HMI tags "2080AG504M01"
   "2080AG504M01.AI1" : Real AT %DB4149.DBD6, 500 ms
   "2080AG504M01.AI2" : Real AT %DB4149.DBD10, 500 ms
   "2080AG504M01.AI3" : Real AT %DB4149.DBD14, 500 ms
   "2080AG504M01.AO1a" : Real AT %DB4149.DBD34, 500 ms
   "2080AG504M01.AO1b" : Real AT %DB4149.DBD38, 500 ms
   "2080AG504M01.AO2a" : Real AT %DB4149.DBD42, 500 ms
   "2080AG504M01.AO2b" : Real AT %DB4149.DBD42, 500 ms
   "2080AG504M01.AO3a" : Real AT %DB4149.DBD50, 500 ms
   "2080AG504M01.AO3b" : Real AT %DB4149.DBD46, 500 ms
   "2080AG504M01.BlockInfo" : Array [0..4] of Int AT %DB4149.DBX74.0, 500 ms
   "2080AG504M01.DefaultText" : TextRef, internal   // Заголовок POPUP окна. При експорте из ECS через скрипт заполняется автоматически, если теги копируются в ручную то требуется в ручную задатать свойство Start Value
   "2080AG504M01.DI.ACK" : Bool AT %DB4149.DBX5.3, 500 ms
   "2080AG504M01.DI.ASTR" : Bool AT %DB4149.DBX2.1, 500 ms
   "2080AG504M01.DI.BUSF" : Bool AT %DB4149.DBX4.5, 500 ms
   "2080AG504M01.DI.DIR" : Bool AT %DB4149.DBX2.2, 500 ms
   "2080AG504M01.DI.DOPR" : Bool AT %DB4149.DBX4.6, 500 ms
   "2080AG504M01.DI.DRDY" : Bool AT %DB4149.DBX3.6, 500 ms
   "2080AG504M01.DI.DTEST" : Bool AT %DB4149.DBX4.7, 500 ms
   "2080AG504M01.DI.EARTH" : Bool AT %DB4149.DBX4.1, 500 ms
   "2080AG504M01.DI.ES" : Bool AT %DB4149.DBX5.2, 500 ms
   "2080AG504M01.DI.GFA" : Bool AT %DB4149.DBX4.3, 500 ms
   "2080AG504M01.DI.GWA" : Bool AT %DB4149.DBX4.4, 500 ms
   "2080AG504M01.DI.LSTP" : Bool AT %DB4149.DBX3.2, 500 ms
   "2080AG504M01.DI.LSTR1" : Bool AT %DB4149.DBX3.0, 500 ms
   "2080AG504M01.DI.LSTR2" : Bool AT %DB4149.DBX3.1, 500 ms
   "2080AG504M01.DI.MCC" : Bool AT %DB4149.DBX2.3, 500 ms
   "2080AG504M01.DI.MD" : Bool AT %DB4149.DBX3.7, 500 ms
   "2080AG504M01.DI.OVL" : Bool AT %DB4149.DBX2.5, 500 ms
   "2080AG504M01.DI.RDY" : Bool AT %DB4149.DBX2.4, 500 ms
   "2080AG504M01.DI.REM" : Bool AT %DB4149.DBX3.3, 500 ms
   "2080AG504M01.DI.RET1" : Bool AT %DB4149.DBX2.6, 500 ms
   "2080AG504M01.DI.RET2" : Bool AT %DB4149.DBX2.7, 500 ms
   "2080AG504M01.DI.SEL" : Bool AT %DB4149.DBX2.0, 500 ms
   "2080AG504M01.DI.SFS" : Bool AT %DB4149.DBX5.0, 500 ms
   "2080AG504M01.DI.SLS" : Bool AT %DB4149.DBX5.1, 500 ms
   "2080AG504M01.DI.SSW" : Bool AT %DB4149.DBX3.4, 500 ms
   "2080AG504M01.DI.STALL" : Bool AT %DB4149.DBX4.0, 500 ms
   "2080AG504M01.DI.TFA" : Bool AT %DB4149.DBX3.5, 500 ms
   "2080AG504M01.DI.UBAL" : Bool AT %DB4149.DBX4.2, 500 ms
   "2080AG504M01.DQ.ASTW" : Bool AT %DB4149.DBX32.0, 500 ms
   "2080AG504M01.DQ.AUT" : Bool AT %DB4149.DBX31.4, 500 ms
   "2080AG504M01.DQ.CON1" : Bool AT %DB4149.DBX30.0, 500 ms
   "2080AG504M01.DQ.CON2" : Bool AT %DB4149.DBX30.1, 500 ms
   "2080AG504M01.DQ.LAMP1" : Bool AT %DB4149.DBX30.2, 500 ms
   "2080AG504M01.DQ.LAMP2" : Bool AT %DB4149.DBX30.3, 500 ms
   "2080AG504M01.DQ.LOC" : Bool AT %DB4149.DBX31.2, 500 ms
   "2080AG504M01.DQ.MAN" : Bool AT %DB4149.DBX31.3, 500 ms
   "2080AG504M01.DQ.OK" : Bool AT %DB4149.DBX31.1, 500 ms
   "2080AG504M01.DQ.RD1" : Bool AT %DB4149.DBX30.5, 500 ms
   "2080AG504M01.DQ.RD2" : Bool AT %DB4149.DBX30.6, 500 ms
   "2080AG504M01.DQ.RES" : Bool AT %DB4149.DBX31.6, 500 ms
   "2080AG504M01.DQ.RUN1" : Bool AT %DB4149.DBX30.7, 500 ms
   "2080AG504M01.DQ.RUN2" : Bool AT %DB4149.DBX31.0, 500 ms
   "2080AG504M01.DQ.SACK" : Bool AT %DB4149.DBX30.4, 500 ms
   "2080AG504M01.DQ.SS" : Bool AT %DB4149.DBX31.5, 500 ms
   "2080AG504M01.DQ.TESTP" : Bool AT %DB4149.DBX31.7, 500 ms
   "2080AG504M01.FP_CMD" : Int AT %DB4149.DBW84, 500 ms
   "2080AG504M01.FP_CMD.AckAlarm" : Bool AT %DB4149.DBX84.7, 500 ms
   "2080AG504M01.FP_CMD.Auto" : Bool AT %DB4149.DBX85.0, 500 ms
   "2080AG504M01.FP_CMD.Local" : Bool AT %DB4149.DBX85.2, 500 ms
   "2080AG504M01.FP_CMD.Manual" : Bool AT %DB4149.DBX85.1, 500 ms
   "2080AG504M01.FP_CMD.QuickStop" : Bool AT %DB4149.DBX84.0, 500 ms
   "2080AG504M01.FP_CMD.Reset" : Bool AT %DB4149.DBX85.6, 500 ms
   "2080AG504M01.FP_CMD.Start1" : Bool AT %DB4149.DBX85.3, 500 ms
   "2080AG504M01.FP_CMD.Start2" : Bool AT %DB4149.DBX85.4, 500 ms
   "2080AG504M01.FP_CMD.Stop" : Bool AT %DB4149.DBX85.5, 500 ms
   "2080AG504M01.FP_CMD.Test" : Bool AT %DB4149.DBX85.7, 500 ms
   "2080AG504M01.FP_DIM.Auto" : Bool AT %DB4149.DBX92.0, 500 ms
   "2080AG504M01.FP_DIM.FP_DIM" : Bool AT %DB4149.DBX92.0, 500 ms
   "2080AG504M01.FP_DIM.Local" : Bool AT %DB4149.DBX92.1, 500 ms
   "2080AG504M01.FP_DIM.Manual" : Bool AT %DB4149.DBX92.2, 500 ms
   "2080AG504M01.FP_DIM.QStop" : Bool AT %DB4149.DBX92.7, 500 ms
   "2080AG504M01.FP_DIM.Reset" : Bool AT %DB4149.DBX93.0, 500 ms
   "2080AG504M01.FP_DIM.Start1" : Bool AT %DB4149.DBX92.3, 500 ms
   "2080AG504M01.FP_DIM.Start2" : Bool AT %DB4149.DBX92.4, 500 ms
   "2080AG504M01.FP_DIM.Stop" : Bool AT %DB4149.DBX92.5, 500 ms
   "2080AG504M01.FP_DIM.TEst" : Bool AT %DB4149.DBX92.6, 500 ms
   "2080AG504M01.FP_DIM1" : Array [0..15] of Bool AT %DB4149.DBX92.0, 500 ms
   "2080AG504M01.FP_EN.Mode_Auto" : Bool AT %DB4149.DBX90.0, 500 ms
   "2080AG504M01.FP_EN.Mode_Loc" : Bool AT %DB4149.DBX90.2, 500 ms
   "2080AG504M01.FP_EN.Mode_Loc_1" : Bool AT %DB4149.DBX90.3, 500 ms
   "2080AG504M01.FP_EN.Mode_Man" : Bool AT %DB4149.DBX90.1, 500 ms
   "2080AG504M01.FP_EN.Mode_SS_Field" : Bool AT %DB4149.DBX90.4, 500 ms
   "2080AG504M01.FP_EN.Mode_SS_FP" : Bool AT %DB4149.DBX90.5, 500 ms
   "2080AG504M01.FP_EN.Mode_Test" : Bool AT %DB4149.DBX90.3, 500 ms
   "2080AG504M01.FP_EN.PB_QStop" : Bool AT %DB4149.DBX90.6, 500 ms
   "2080AG504M01.FP_PARM.AI1_Max" : Real AT %DB4149.DBD158, 500 ms
   "2080AG504M01.FP_PARM.AI1_Min" : Real AT %DB4149.DBD162, 500 ms
   "2080AG504M01.FP_PARM.AI2_Max" : Real AT %DB4149.DBD166, 500 ms
   "2080AG504M01.FP_PARM.AI2_Min" : Real AT %DB4149.DBD170, 500 ms
   "2080AG504M01.FP_PARM.AI3_Max" : Real AT %DB4149.DBD174, 500 ms
   "2080AG504M01.FP_PARM.AI3_Min" : Real AT %DB4149.DBD178, 500 ms
   "2080AG504M01.FP_PARM.AO1a_Max" : Real AT %DB4149.DBD182, 500 ms
   "2080AG504M01.FP_PARM.AO1a_Min" : Real AT %DB4149.DBD186, 500 ms
   "2080AG504M01.FP_PARM.AO1b_Max" : Real AT %DB4149.DBD206, 500 ms
   "2080AG504M01.FP_PARM.AO1b_Min" : Real AT %DB4149.DBD210, 500 ms
   "2080AG504M01.FP_PARM.AO2a_Max" : Real AT %DB4149.DBD190, 500 ms
   "2080AG504M01.FP_PARM.AO2a_Min" : Real AT %DB4149.DBD194, 500 ms
   "2080AG504M01.FP_PARM.AO2b_Max" : Real AT %DB4149.DBD214, 500 ms
   "2080AG504M01.FP_PARM.AO2b_Min" : Real AT %DB4149.DBD218, 500 ms
   "2080AG504M01.FP_PARM.AO3a_Max" : Real AT %DB4149.DBD198, 500 ms
   "2080AG504M01.FP_PARM.AO3a_Min" : Real AT %DB4149.DBD202, 500 ms
   "2080AG504M01.FP_PARM.AO3b_Max" : Real AT %DB4149.DBD222, 500 ms
   "2080AG504M01.FP_PARM.AO3b_Min" : Real AT %DB4149.DBD226, 500 ms
   "2080AG504M01.FP_PARM.ChangeDir_Acc" : Int AT %DB4149.DBW138, 500 ms
   "2080AG504M01.FP_PARM.ChangeDir_Pre" : Int AT %DB4149.DBW136, 500 ms
   "2080AG504M01.FP_PARM.DelayStart_Acc" : Int AT %DB4149.DBW114, 500 ms
   "2080AG504M01.FP_PARM.DelayStart_Pre" : Int AT %DB4149.DBW112, 500 ms
   "2080AG504M01.FP_PARM.DelayStop_Acc" : Int AT %DB4149.DBW118, 500 ms
   "2080AG504M01.FP_PARM.DelayStop_Pre" : Int AT %DB4149.DBW116, 500 ms
   "2080AG504M01.FP_PARM.INTL" : Bool AT %DB4149.DBX230.0, 500 ms
   "2080AG504M01.FP_PARM.INTL_SEQ_STP" : Bool AT %DB4149.DBX230.3, 500 ms
   "2080AG504M01.FP_PARM.INTL_SEQ_STR1" : Bool AT %DB4149.DBX230.1, 500 ms
   "2080AG504M01.FP_PARM.INTL_SEQ_STR2" : Bool AT %DB4149.DBX230.2, 500 ms
   "2080AG504M01.FP_PARM.LeaveFS_Acc" : Int AT %DB4149.DBW142, 500 ms
   "2080AG504M01.FP_PARM.LeaveFS_Pre" : Int AT %DB4149.DBW140, 500 ms
   "2080AG504M01.FP_PARM.MD_Freq_PV" : Int AT %DB4149.DBW154, 500 ms
   "2080AG504M01.FP_PARM.MD_Freq_SP" : Int AT %DB4149.DBW152, 500 ms
   "2080AG504M01.FP_PARM.ReachFS_Acc" : Int AT %DB4149.DBW150, 500 ms
   "2080AG504M01.FP_PARM.ReachFS_Pre" : Int AT %DB4149.DBW148, 500 ms
   "2080AG504M01.FP_PARM.ReachLS_Acc" : Int AT %DB4149.DBW146, 500 ms
   "2080AG504M01.FP_PARM.ReachLS_Pre" : Int AT %DB4149.DBW144, 500 ms
   "2080AG504M01.FP_PARM.ReturnMon_Acc" : Int AT %DB4149.DBW122, 500 ms
   "2080AG504M01.FP_PARM.ReturnMon_Pre" : Int AT %DB4149.DBW120, 500 ms
   "2080AG504M01.FP_PARM.RunDelay1_Acc" : Int AT %DB4149.DBW106, 500 ms
   "2080AG504M01.FP_PARM.RunDelay1_Pre" : Int AT %DB4149.DBW104, 500 ms
   "2080AG504M01.FP_PARM.RunDelay2_Acc" : Int AT %DB4149.DBW110, 500 ms
   "2080AG504M01.FP_PARM.RunDelay2_Pre" : Int AT %DB4149.DBW108, 500 ms
   "2080AG504M01.FP_PARM.SpeedMonOffDelay_Acc" : Int AT %DB4149.DBW130, 500 ms
   "2080AG504M01.FP_PARM.SpeedMonOffDelay_Pre" : Int AT %DB4149.DBW128, 500 ms
   "2080AG504M01.FP_PARM.SpeedMonOnDelay_Acc" : Int AT %DB4149.DBW126, 500 ms
   "2080AG504M01.FP_PARM.SpeedMonOnDelay_Pre" : Int AT %DB4149.DBW124, 500 ms
   "2080AG504M01.FP_PARM.SpeedMonTrigDelay_Acc" : Int AT %DB4149.DBW134, 500 ms
   "2080AG504M01.FP_PARM.SpeedMonTrigDelay_Pre" : Int AT %DB4149.DBW132, 500 ms
   "2080AG504M01.FP_PARM.StartWarn_Acc" : Int AT %DB4149.DBW102, 500 ms
   "2080AG504M01.FP_PARM.StartWarn_Pre" : Int AT %DB4149.DBW100, 500 ms
   "2080AG504M01.FP_PARM.StopReason" : Int AT %DB4149.DBW156, 500 ms
   "2080AG504M01.FP_SEL.INCH_Loc" : Bool AT %DB4149.DBX87.7, 500 ms
   "2080AG504M01.FP_SEL.INCH_Man" : Bool AT %DB4149.DBX87.6, 500 ms
   "2080AG504M01.FP_SEL.MD" : Bool AT %DB4149.DBX86.0, 500 ms
   "2080AG504M01.FP_SEL.MD_Maintain" : Bool AT %DB4149.DBX86.3, 500 ms
   "2080AG504M01.FP_SEL.MD_OnOff" : Bool AT %DB4149.DBX86.2, 500 ms
   "2080AG504M01.FP_SEL.MD_Puls" : Bool AT %DB4149.DBX86.1, 500 ms
   "2080AG504M01.FP_SEL.MotorStarter" : Bool AT %DB4149.DBX87.3, 500 ms
   "2080AG504M01.FP_SEL.OutOfSevice" : Bool AT %DB4149.DBX88.0, 500 ms
   "2080AG504M01.FP_SEL.ParentCollection" : Bool AT %DB4149.DBX87.5, 500 ms
   "2080AG504M01.FP_SEL.ParentSupress" : Bool AT %DB4149.DBX87.4, 500 ms
   "2080AG504M01.FP_SEL.STW_AutoStart" : Bool AT %DB4149.DBX86.4, 500 ms
   "2080AG504M01.FP_SEL.STW_Local" : Bool AT %DB4149.DBX86.5, 500 ms
   "2080AG504M01.FP_SEL.STW_Manual" : Bool AT %DB4149.DBX86.6, 500 ms
   "2080AG504M01.FP_SEL.STW_Single" : Bool AT %DB4149.DBX86.7, 500 ms
   "2080AG504M01.FP_SEL.Type_Bimotor" : Bool AT %DB4149.DBX87.1, 500 ms
   "2080AG504M01.FP_SEL.Type_Indication" : Bool AT %DB4149.DBX87.2, 500 ms
   "2080AG504M01.FP_SEL.Type_Unimotor" : Bool AT %DB4149.DBX87.0, 500 ms
   "2080AG504M01.FP_SEL.WarningDrive" : Bool AT %DB4149.DBX88.1, 500 ms
   "2080AG504M01.FP_SHOW.ACK" : Bool AT %DB4149.DBX97.5, 500 ms
   "2080AG504M01.FP_SHOW.AI1" : Bool AT %DB4149.DBX95.0, 500 ms
   "2080AG504M01.FP_SHOW.AI2" : Bool AT %DB4149.DBX95.1, 500 ms
   "2080AG504M01.FP_SHOW.AI3" : Bool AT %DB4149.DBX95.2, 500 ms
   "2080AG504M01.FP_SHOW.ASTR" : Bool AT %DB4149.DBX99.2, 500 ms
   "2080AG504M01.FP_SHOW.B1" : Byte AT %DB4149.DBB95, 500 ms
   "2080AG504M01.FP_SHOW.B2" : Byte AT %DB4149.DBB96, 500 ms
   "2080AG504M01.FP_SHOW.B3" : Byte AT %DB4149.DBB97, 500 ms
   "2080AG504M01.FP_SHOW.B4" : Byte AT %DB4149.DBB98, 500 ms
   "2080AG504M01.FP_SHOW.BUSF" : Bool AT %DB4149.DBX97.2, 500 ms
   "2080AG504M01.FP_SHOW.ChangeDir" : Bool AT %DB4149.DBX99.0, 500 ms
   "2080AG504M01.FP_SHOW.CON2" : Bool AT %DB4149.DBX98.2, 500 ms
   "2080AG504M01.FP_SHOW.DelayRun2" : Bool AT %DB4149.DBX98.7, 500 ms
   "2080AG504M01.FP_SHOW.DOPR" : Bool AT %DB4149.DBX97.3, 500 ms
   "2080AG504M01.FP_SHOW.DRDY" : Bool AT %DB4149.DBX96.4, 500 ms
   "2080AG504M01.FP_SHOW.DTEST" : Bool AT %DB4149.DBX97.4, 500 ms
   "2080AG504M01.FP_SHOW.EARTH" : Bool AT %DB4149.DBX96.6, 500 ms
   "2080AG504M01.FP_SHOW.ES" : Bool AT %DB4149.DBX96.2, 500 ms
   "2080AG504M01.FP_SHOW.GFA" : Bool AT %DB4149.DBX97.0, 500 ms
   "2080AG504M01.FP_SHOW.GWA" : Bool AT %DB4149.DBX97.1, 500 ms
   "2080AG504M01.FP_SHOW.LSTP" : Bool AT %DB4149.DBX95.7, 500 ms
   "2080AG504M01.FP_SHOW.LSTR1" : Bool AT %DB4149.DBX97.6, 500 ms
   "2080AG504M01.FP_SHOW.LSTR2" : Bool AT %DB4149.DBX97.7, 500 ms
   "2080AG504M01.FP_SHOW.MCC" : Bool AT %DB4149.DBX95.4, 500 ms
   "2080AG504M01.FP_SHOW.MD" : Bool AT %DB4149.DBX98.6, 500 ms
   "2080AG504M01.FP_SHOW.OVL" : Bool AT %DB4149.DBX95.6, 500 ms
   "2080AG504M01.FP_SHOW.PB_Auto" : Bool AT %DB4149.DBX94.0, 500 ms
   "2080AG504M01.FP_SHOW.PB_Local" : Bool AT %DB4149.DBX94.1, 500 ms
   "2080AG504M01.FP_SHOW.PB_Manual" : Bool AT %DB4149.DBX94.2, 500 ms
   "2080AG504M01.FP_SHOW.PB_QStop" : Bool AT %DB4149.DBX94.7, 500 ms
   "2080AG504M01.FP_SHOW.PB_Reset" : Bool AT %DB4149.DBX99.1, 500 ms
   "2080AG504M01.FP_SHOW.PB_Start1" : Bool AT %DB4149.DBX94.3, 500 ms
   "2080AG504M01.FP_SHOW.PB_Start2" : Bool AT %DB4149.DBX94.4, 500 ms
   "2080AG504M01.FP_SHOW.PB_Stop" : Bool AT %DB4149.DBX94.5, 500 ms
   "2080AG504M01.FP_SHOW.PB_Test" : Bool AT %DB4149.DBX94.6, 500 ms
   "2080AG504M01.FP_SHOW.RD2" : Bool AT %DB4149.DBX98.3, 500 ms
   "2080AG504M01.FP_SHOW.RDY" : Bool AT %DB4149.DBX95.5, 500 ms
   "2080AG504M01.FP_SHOW.REM" : Bool AT %DB4149.DBX96.0, 500 ms
   "2080AG504M01.FP_SHOW.RET2" : Bool AT %DB4149.DBX98.0, 500 ms
   "2080AG504M01.FP_SHOW.RUN2" : Bool AT %DB4149.DBX98.1, 500 ms
   "2080AG504M01.FP_SHOW.SFS" : Bool AT %DB4149.DBX98.4, 500 ms
   "2080AG504M01.FP_SHOW.SLS" : Bool AT %DB4149.DBX98.5, 500 ms
   "2080AG504M01.FP_SHOW.SP" : Bool AT %DB4149.DBX95.3, 500 ms
   "2080AG504M01.FP_SHOW.SSW" : Bool AT %DB4149.DBX96.1, 500 ms
   "2080AG504M01.FP_SHOW.STALL" : Bool AT %DB4149.DBX96.5, 500 ms
   "2080AG504M01.FP_SHOW.TFA" : Bool AT %DB4149.DBX96.3, 500 ms
   "2080AG504M01.FP_SHOW.UBAL" : Bool AT %DB4149.DBX96.7, 500 ms
   "2080AG504M01.ModePointer" : Int AT %DB4149.DBW496, 500 ms
   "2080AG504M01.MSW" : DWord AT %DB4149.DBD62, 500 ms
   "2080AG504M01.ParentInfo" : TextRef, internal   // Имя родителя для попап окна, вкладка инфо. При експорте из ECS через скрипт заполняется автоматически, если теги копируются в ручную то требуется в ручную задатать свойство Start Value
   "2080AG504M01.SPSET" : Real AT %DB4149.DBD18, 500 ms
   "2080AG504M01.StatusWork" : Int AT %DB4149.DBW494, 500 ms
   "2080AG504M01.STR01" : Byte AT %DB10.DBB103, 500 ms   // Interlock
   "2080AG504M01.STR01.DefaultText" : TextRef, internal
   "2080AG504M01.STR02" : Byte AT %DB10.DBB104, 500 ms   // Interlock
   "2080AG504M01.STR02.DefaultText" : TextRef, internal
   "2080AG504M01.STR03" : Byte AT %DB10.DBB105, 500 ms   // Interlock
   "2080AG504M01.STR03.DefaultText" : TextRef, internal
   "2080AG504M01.STR04" : Byte AT %DB10.DBB106, 500 ms   // Interlock
   "2080AG504M01.STR04.DefaultText" : TextRef, internal

HMI tags "2080AG505M01"
   "2080AG505M01.AI1" : Real AT %DB4151.DBD6, 500 ms
   "2080AG505M01.AI2" : Real AT %DB4151.DBD10, 500 ms
   "2080AG505M01.AI3" : Real AT %DB4151.DBD14, 500 ms
   "2080AG505M01.AO1a" : Real AT %DB4151.DBD34, 500 ms
   "2080AG505M01.AO1b" : Real AT %DB4151.DBD38, 500 ms
   "2080AG505M01.AO2a" : Real AT %DB4151.DBD42, 500 ms
   "2080AG505M01.AO2b" : Real AT %DB4151.DBD42, 500 ms
   "2080AG505M01.AO3a" : Real AT %DB4151.DBD50, 500 ms
   "2080AG505M01.AO3b" : Real AT %DB4151.DBD46, 500 ms
   "2080AG505M01.BlockInfo" : Array [0..4] of Int AT %DB4151.DBX74.0, 500 ms
   "2080AG505M01.DefaultText" : TextRef, internal   // Заголовок POPUP окна. При експорте из ECS через скрипт заполняется автоматически, если теги копируются в ручную то требуется в ручную задатать свойство Start Value
   "2080AG505M01.DI.ACK" : Bool AT %DB4151.DBX5.3, 500 ms
   "2080AG505M01.DI.ASTR" : Bool AT %DB4151.DBX2.1, 500 ms
   "2080AG505M01.DI.BUSF" : Bool AT %DB4151.DBX4.5, 500 ms
   "2080AG505M01.DI.DIR" : Bool AT %DB4151.DBX2.2, 500 ms
   "2080AG505M01.DI.DOPR" : Bool AT %DB4151.DBX4.6, 500 ms
   "2080AG505M01.DI.DRDY" : Bool AT %DB4151.DBX3.6, 500 ms
   "2080AG505M01.DI.DTEST" : Bool AT %DB4151.DBX4.7, 500 ms
   "2080AG505M01.DI.EARTH" : Bool AT %DB4151.DBX4.1, 500 ms
   "2080AG505M01.DI.ES" : Bool AT %DB4151.DBX5.2, 500 ms
   "2080AG505M01.DI.GFA" : Bool AT %DB4151.DBX4.3, 500 ms
   "2080AG505M01.DI.GWA" : Bool AT %DB4151.DBX4.4, 500 ms
   "2080AG505M01.DI.LSTP" : Bool AT %DB4151.DBX3.2, 500 ms
   "2080AG505M01.DI.LSTR1" : Bool AT %DB4151.DBX3.0, 500 ms
   "2080AG505M01.DI.LSTR2" : Bool AT %DB4151.DBX3.1, 500 ms
   "2080AG505M01.DI.MCC" : Bool AT %DB4151.DBX2.3, 500 ms
   "2080AG505M01.DI.MD" : Bool AT %DB4151.DBX3.7, 500 ms
   "2080AG505M01.DI.OVL" : Bool AT %DB4151.DBX2.5, 500 ms
   "2080AG505M01.DI.RDY" : Bool AT %DB4151.DBX2.4, 500 ms
   "2080AG505M01.DI.REM" : Bool AT %DB4151.DBX3.3, 500 ms
   "2080AG505M01.DI.RET1" : Bool AT %DB4151.DBX2.6, 500 ms
   "2080AG505M01.DI.RET2" : Bool AT %DB4151.DBX2.7, 500 ms
   "2080AG505M01.DI.SEL" : Bool AT %DB4151.DBX2.0, 500 ms
   "2080AG505M01.DI.SFS" : Bool AT %DB4151.DBX5.0, 500 ms
   "2080AG505M01.DI.SLS" : Bool AT %DB4151.DBX5.1, 500 ms
   "2080AG505M01.DI.SSW" : Bool AT %DB4151.DBX3.4, 500 ms
   "2080AG505M01.DI.STALL" : Bool AT %DB4151.DBX4.0, 500 ms
   "2080AG505M01.DI.TFA" : Bool AT %DB4151.DBX3.5, 500 ms
   "2080AG505M01.DI.UBAL" : Bool AT %DB4151.DBX4.2, 500 ms
   "2080AG505M01.DQ.ASTW" : Bool AT %DB4151.DBX32.0, 500 ms
   "2080AG505M01.DQ.AUT" : Bool AT %DB4151.DBX31.4, 500 ms
   "2080AG505M01.DQ.CON1" : Bool AT %DB4151.DBX30.0, 500 ms
   "2080AG505M01.DQ.CON2" : Bool AT %DB4151.DBX30.1, 500 ms
   "2080AG505M01.DQ.LAMP1" : Bool AT %DB4151.DBX30.2, 500 ms
   "2080AG505M01.DQ.LAMP2" : Bool AT %DB4151.DBX30.3, 500 ms
   "2080AG505M01.DQ.LOC" : Bool AT %DB4151.DBX31.2, 500 ms
   "2080AG505M01.DQ.MAN" : Bool AT %DB4151.DBX31.3, 500 ms
   "2080AG505M01.DQ.OK" : Bool AT %DB4151.DBX31.1, 500 ms
   "2080AG505M01.DQ.RD1" : Bool AT %DB4151.DBX30.5, 500 ms
   "2080AG505M01.DQ.RD2" : Bool AT %DB4151.DBX30.6, 500 ms
   "2080AG505M01.DQ.RES" : Bool AT %DB4151.DBX31.6, 500 ms
   "2080AG505M01.DQ.RUN1" : Bool AT %DB4151.DBX30.7, 500 ms
   "2080AG505M01.DQ.RUN2" : Bool AT %DB4151.DBX31.0, 500 ms
   "2080AG505M01.DQ.SACK" : Bool AT %DB4151.DBX30.4, 500 ms
   "2080AG505M01.DQ.SS" : Bool AT %DB4151.DBX31.5, 500 ms
   "2080AG505M01.DQ.TESTP" : Bool AT %DB4151.DBX31.7, 500 ms
   "2080AG505M01.FP_CMD" : Int AT %DB4151.DBW84, 500 ms
   "2080AG505M01.FP_CMD.AckAlarm" : Bool AT %DB4151.DBX84.7, 500 ms
   "2080AG505M01.FP_CMD.Auto" : Bool AT %DB4151.DBX85.0, 500 ms
   "2080AG505M01.FP_CMD.Local" : Bool AT %DB4151.DBX85.2, 500 ms
   "2080AG505M01.FP_CMD.Manual" : Bool AT %DB4151.DBX85.1, 500 ms
   "2080AG505M01.FP_CMD.QuickStop" : Bool AT %DB4151.DBX84.0, 500 ms
   "2080AG505M01.FP_CMD.Reset" : Bool AT %DB4151.DBX85.6, 500 ms
   "2080AG505M01.FP_CMD.Start1" : Bool AT %DB4151.DBX85.3, 500 ms
   "2080AG505M01.FP_CMD.Start2" : Bool AT %DB4151.DBX85.4, 500 ms
   "2080AG505M01.FP_CMD.Stop" : Bool AT %DB4151.DBX85.5, 500 ms
   "2080AG505M01.FP_CMD.Test" : Bool AT %DB4151.DBX85.7, 500 ms
   "2080AG505M01.FP_DIM.Auto" : Bool AT %DB4151.DBX92.0, 500 ms
   "2080AG505M01.FP_DIM.FP_DIM" : Bool AT %DB4151.DBX92.0, 500 ms
   "2080AG505M01.FP_DIM.Local" : Bool AT %DB4151.DBX92.1, 500 ms
   "2080AG505M01.FP_DIM.Manual" : Bool AT %DB4151.DBX92.2, 500 ms
   "2080AG505M01.FP_DIM.QStop" : Bool AT %DB4151.DBX92.7, 500 ms
   "2080AG505M01.FP_DIM.Reset" : Bool AT %DB4151.DBX93.0, 500 ms
   "2080AG505M01.FP_DIM.Start1" : Bool AT %DB4151.DBX92.3, 500 ms
   "2080AG505M01.FP_DIM.Start2" : Bool AT %DB4151.DBX92.4, 500 ms
   "2080AG505M01.FP_DIM.Stop" : Bool AT %DB4151.DBX92.5, 500 ms
   "2080AG505M01.FP_DIM.TEst" : Bool AT %DB4151.DBX92.6, 500 ms
   "2080AG505M01.FP_DIM1" : Array [0..15] of Bool AT %DB4151.DBX92.0, 500 ms
   "2080AG505M01.FP_EN.Mode_Auto" : Bool AT %DB4151.DBX90.0, 500 ms
   "2080AG505M01.FP_EN.Mode_Loc" : Bool AT %DB4151.DBX90.2, 500 ms
   "2080AG505M01.FP_EN.Mode_Loc_1" : Bool AT %DB4151.DBX90.3, 500 ms
   "2080AG505M01.FP_EN.Mode_Man" : Bool AT %DB4151.DBX90.1, 500 ms
   "2080AG505M01.FP_EN.Mode_SS_Field" : Bool AT %DB4151.DBX90.4, 500 ms
   "2080AG505M01.FP_EN.Mode_SS_FP" : Bool AT %DB4151.DBX90.5, 500 ms
   "2080AG505M01.FP_EN.Mode_Test" : Bool AT %DB4151.DBX90.3, 500 ms
   "2080AG505M01.FP_EN.PB_QStop" : Bool AT %DB4151.DBX90.6, 500 ms
   "2080AG505M01.FP_PARM.AI1_Max" : Real AT %DB4151.DBD158, 500 ms
   "2080AG505M01.FP_PARM.AI1_Min" : Real AT %DB4151.DBD162, 500 ms
   "2080AG505M01.FP_PARM.AI2_Max" : Real AT %DB4151.DBD166, 500 ms
   "2080AG505M01.FP_PARM.AI2_Min" : Real AT %DB4151.DBD170, 500 ms
   "2080AG505M01.FP_PARM.AI3_Max" : Real AT %DB4151.DBD174, 500 ms
   "2080AG505M01.FP_PARM.AI3_Min" : Real AT %DB4151.DBD178, 500 ms
   "2080AG505M01.FP_PARM.AO1a_Max" : Real AT %DB4151.DBD182, 500 ms
   "2080AG505M01.FP_PARM.AO1a_Min" : Real AT %DB4151.DBD186, 500 ms
   "2080AG505M01.FP_PARM.AO1b_Max" : Real AT %DB4151.DBD206, 500 ms
   "2080AG505M01.FP_PARM.AO1b_Min" : Real AT %DB4151.DBD210, 500 ms
   "2080AG505M01.FP_PARM.AO2a_Max" : Real AT %DB4151.DBD190, 500 ms
   "2080AG505M01.FP_PARM.AO2a_Min" : Real AT %DB4151.DBD194, 500 ms
   "2080AG505M01.FP_PARM.AO2b_Max" : Real AT %DB4151.DBD214, 500 ms
   "2080AG505M01.FP_PARM.AO2b_Min" : Real AT %DB4151.DBD218, 500 ms
   "2080AG505M01.FP_PARM.AO3a_Max" : Real AT %DB4151.DBD198, 500 ms
   "2080AG505M01.FP_PARM.AO3a_Min" : Real AT %DB4151.DBD202, 500 ms
   "2080AG505M01.FP_PARM.AO3b_Max" : Real AT %DB4151.DBD222, 500 ms
   "2080AG505M01.FP_PARM.AO3b_Min" : Real AT %DB4151.DBD226, 500 ms
   "2080AG505M01.FP_PARM.ChangeDir_Acc" : Int AT %DB4151.DBW138, 500 ms
   "2080AG505M01.FP_PARM.ChangeDir_Pre" : Int AT %DB4151.DBW136, 500 ms
   "2080AG505M01.FP_PARM.DelayStart_Acc" : Int AT %DB4151.DBW114, 500 ms
   "2080AG505M01.FP_PARM.DelayStart_Pre" : Int AT %DB4151.DBW112, 500 ms
   "2080AG505M01.FP_PARM.DelayStop_Acc" : Int AT %DB4151.DBW118, 500 ms
   "2080AG505M01.FP_PARM.DelayStop_Pre" : Int AT %DB4151.DBW116, 500 ms
   "2080AG505M01.FP_PARM.INTL" : Bool AT %DB4151.DBX230.0, 500 ms
   "2080AG505M01.FP_PARM.INTL_SEQ_STP" : Bool AT %DB4151.DBX230.3, 500 ms
   "2080AG505M01.FP_PARM.INTL_SEQ_STR1" : Bool AT %DB4151.DBX230.1, 500 ms
   "2080AG505M01.FP_PARM.INTL_SEQ_STR2" : Bool AT %DB4151.DBX230.2, 500 ms
   "2080AG505M01.FP_PARM.LeaveFS_Acc" : Int AT %DB4151.DBW142, 500 ms
   "2080AG505M01.FP_PARM.LeaveFS_Pre" : Int AT %DB4151.DBW140, 500 ms
   "2080AG505M01.FP_PARM.MD_Freq_PV" : Int AT %DB4151.DBW154, 500 ms
   "2080AG505M01.FP_PARM.MD_Freq_SP" : Int AT %DB4151.DBW152, 500 ms
   "2080AG505M01.FP_PARM.ReachFS_Acc" : Int AT %DB4151.DBW150, 500 ms
   "2080AG505M01.FP_PARM.ReachFS_Pre" : Int AT %DB4151.DBW148, 500 ms
   "2080AG505M01.FP_PARM.ReachLS_Acc" : Int AT %DB4151.DBW146, 500 ms
   "2080AG505M01.FP_PARM.ReachLS_Pre" : Int AT %DB4151.DBW144, 500 ms
   "2080AG505M01.FP_PARM.ReturnMon_Acc" : Int AT %DB4151.DBW122, 500 ms
   "2080AG505M01.FP_PARM.ReturnMon_Pre" : Int AT %DB4151.DBW120, 500 ms
   "2080AG505M01.FP_PARM.RunDelay1_Acc" : Int AT %DB4151.DBW106, 500 ms
   "2080AG505M01.FP_PARM.RunDelay1_Pre" : Int AT %DB4151.DBW104, 500 ms
   "2080AG505M01.FP_PARM.RunDelay2_Acc" : Int AT %DB4151.DBW110, 500 ms
   "2080AG505M01.FP_PARM.RunDelay2_Pre" : Int AT %DB4151.DBW108, 500 ms
   "2080AG505M01.FP_PARM.SpeedMonOffDelay_Acc" : Int AT %DB4151.DBW130, 500 ms
   "2080AG505M01.FP_PARM.SpeedMonOffDelay_Pre" : Int AT %DB4151.DBW128, 500 ms
   "2080AG505M01.FP_PARM.SpeedMonOnDelay_Acc" : Int AT %DB4151.DBW126, 500 ms
   "2080AG505M01.FP_PARM.SpeedMonOnDelay_Pre" : Int AT %DB4151.DBW124, 500 ms
   "2080AG505M01.FP_PARM.SpeedMonTrigDelay_Acc" : Int AT %DB4151.DBW134, 500 ms
   "2080AG505M01.FP_PARM.SpeedMonTrigDelay_Pre" : Int AT %DB4151.DBW132, 500 ms
   "2080AG505M01.FP_PARM.StartWarn_Acc" : Int AT %DB4151.DBW102, 500 ms
   "2080AG505M01.FP_PARM.StartWarn_Pre" : Int AT %DB4151.DBW100, 500 ms
   "2080AG505M01.FP_PARM.StopReason" : Int AT %DB4151.DBW156, 500 ms
   "2080AG505M01.FP_SEL.INCH_Loc" : Bool AT %DB4151.DBX87.7, 500 ms
   "2080AG505M01.FP_SEL.INCH_Man" : Bool AT %DB4151.DBX87.6, 500 ms
   "2080AG505M01.FP_SEL.MD" : Bool AT %DB4151.DBX86.0, 500 ms
   "2080AG505M01.FP_SEL.MD_Maintain" : Bool AT %DB4151.DBX86.3, 500 ms
   "2080AG505M01.FP_SEL.MD_OnOff" : Bool AT %DB4151.DBX86.2, 500 ms
   "2080AG505M01.FP_SEL.MD_Puls" : Bool AT %DB4151.DBX86.1, 500 ms
   "2080AG505M01.FP_SEL.MotorStarter" : Bool AT %DB4151.DBX87.3, 500 ms
   "2080AG505M01.FP_SEL.OutOfSevice" : Bool AT %DB4151.DBX88.0, 500 ms
   "2080AG505M01.FP_SEL.ParentCollection" : Bool AT %DB4151.DBX87.5, 500 ms
   "2080AG505M01.FP_SEL.ParentSupress" : Bool AT %DB4151.DBX87.4, 500 ms
   "2080AG505M01.FP_SEL.STW_AutoStart" : Bool AT %DB4151.DBX86.4, 500 ms
   "2080AG505M01.FP_SEL.STW_Local" : Bool AT %DB4151.DBX86.5, 500 ms
   "2080AG505M01.FP_SEL.STW_Manual" : Bool AT %DB4151.DBX86.6, 500 ms
   "2080AG505M01.FP_SEL.STW_Single" : Bool AT %DB4151.DBX86.7, 500 ms
   "2080AG505M01.FP_SEL.Type_Bimotor" : Bool AT %DB4151.DBX87.1, 500 ms
   "2080AG505M01.FP_SEL.Type_Indication" : Bool AT %DB4151.DBX87.2, 500 ms
   "2080AG505M01.FP_SEL.Type_Unimotor" : Bool AT %DB4151.DBX87.0, 500 ms
   "2080AG505M01.FP_SEL.WarningDrive" : Bool AT %DB4151.DBX88.1, 500 ms
   "2080AG505M01.FP_SHOW.ACK" : Bool AT %DB4151.DBX97.5, 500 ms
   "2080AG505M01.FP_SHOW.AI1" : Bool AT %DB4151.DBX95.0, 500 ms
   "2080AG505M01.FP_SHOW.AI2" : Bool AT %DB4151.DBX95.1, 500 ms
   "2080AG505M01.FP_SHOW.AI3" : Bool AT %DB4151.DBX95.2, 500 ms
   "2080AG505M01.FP_SHOW.ASTR" : Bool AT %DB4151.DBX99.2, 500 ms
   "2080AG505M01.FP_SHOW.B1" : Byte AT %DB4151.DBB95, 500 ms
   "2080AG505M01.FP_SHOW.B2" : Byte AT %DB4151.DBB96, 500 ms
   "2080AG505M01.FP_SHOW.B3" : Byte AT %DB4151.DBB97, 500 ms
   "2080AG505M01.FP_SHOW.B4" : Byte AT %DB4151.DBB98, 500 ms
   "2080AG505M01.FP_SHOW.BUSF" : Bool AT %DB4151.DBX97.2, 500 ms
   "2080AG505M01.FP_SHOW.ChangeDir" : Bool AT %DB4151.DBX99.0, 500 ms
   "2080AG505M01.FP_SHOW.CON2" : Bool AT %DB4151.DBX98.2, 500 ms
   "2080AG505M01.FP_SHOW.DelayRun2" : Bool AT %DB4151.DBX98.7, 500 ms
   "2080AG505M01.FP_SHOW.DOPR" : Bool AT %DB4151.DBX97.3, 500 ms
   "2080AG505M01.FP_SHOW.DRDY" : Bool AT %DB4151.DBX96.4, 500 ms
   "2080AG505M01.FP_SHOW.DTEST" : Bool AT %DB4151.DBX97.4, 500 ms
   "2080AG505M01.FP_SHOW.EARTH" : Bool AT %DB4151.DBX96.6, 500 ms
   "2080AG505M01.FP_SHOW.ES" : Bool AT %DB4151.DBX96.2, 500 ms
   "2080AG505M01.FP_SHOW.GFA" : Bool AT %DB4151.DBX97.0, 500 ms
   "2080AG505M01.FP_SHOW.GWA" : Bool AT %DB4151.DBX97.1, 500 ms
   "2080AG505M01.FP_SHOW.LSTP" : Bool AT %DB4151.DBX95.7, 500 ms
   "2080AG505M01.FP_SHOW.LSTR1" : Bool AT %DB4151.DBX97.6, 500 ms
   "2080AG505M01.FP_SHOW.LSTR2" : Bool AT %DB4151.DBX97.7, 500 ms
   "2080AG505M01.FP_SHOW.MCC" : Bool AT %DB4151.DBX95.4, 500 ms
   "2080AG505M01.FP_SHOW.MD" : Bool AT %DB4151.DBX98.6, 500 ms
   "2080AG505M01.FP_SHOW.OVL" : Bool AT %DB4151.DBX95.6, 500 ms
   "2080AG505M01.FP_SHOW.PB_Auto" : Bool AT %DB4151.DBX94.0, 500 ms
   "2080AG505M01.FP_SHOW.PB_Local" : Bool AT %DB4151.DBX94.1, 500 ms
   "2080AG505M01.FP_SHOW.PB_Manual" : Bool AT %DB4151.DBX94.2, 500 ms
   "2080AG505M01.FP_SHOW.PB_QStop" : Bool AT %DB4151.DBX94.7, 500 ms
   "2080AG505M01.FP_SHOW.PB_Reset" : Bool AT %DB4151.DBX99.1, 500 ms
   "2080AG505M01.FP_SHOW.PB_Start1" : Bool AT %DB4151.DBX94.3, 500 ms
   "2080AG505M01.FP_SHOW.PB_Start2" : Bool AT %DB4151.DBX94.4, 500 ms
   "2080AG505M01.FP_SHOW.PB_Stop" : Bool AT %DB4151.DBX94.5, 500 ms
   "2080AG505M01.FP_SHOW.PB_Test" : Bool AT %DB4151.DBX94.6, 500 ms
   "2080AG505M01.FP_SHOW.RD2" : Bool AT %DB4151.DBX98.3, 500 ms
   "2080AG505M01.FP_SHOW.RDY" : Bool AT %DB4151.DBX95.5, 500 ms
   "2080AG505M01.FP_SHOW.REM" : Bool AT %DB4151.DBX96.0, 500 ms
   "2080AG505M01.FP_SHOW.RET2" : Bool AT %DB4151.DBX98.0, 500 ms
   "2080AG505M01.FP_SHOW.RUN2" : Bool AT %DB4151.DBX98.1, 500 ms
   "2080AG505M01.FP_SHOW.SFS" : Bool AT %DB4151.DBX98.4, 500 ms
   "2080AG505M01.FP_SHOW.SLS" : Bool AT %DB4151.DBX98.5, 500 ms
   "2080AG505M01.FP_SHOW.SP" : Bool AT %DB4151.DBX95.3, 500 ms
   "2080AG505M01.FP_SHOW.SSW" : Bool AT %DB4151.DBX96.1, 500 ms
   "2080AG505M01.FP_SHOW.STALL" : Bool AT %DB4151.DBX96.5, 500 ms
   "2080AG505M01.FP_SHOW.TFA" : Bool AT %DB4151.DBX96.3, 500 ms
   "2080AG505M01.FP_SHOW.UBAL" : Bool AT %DB4151.DBX96.7, 500 ms
   "2080AG505M01.ModePointer" : Int AT %DB4151.DBW496, 500 ms
   "2080AG505M01.MSW" : DWord AT %DB4151.DBD62, 500 ms
   "2080AG505M01.ParentInfo" : TextRef, internal   // Имя родителя для попап окна, вкладка инфо. При експорте из ECS через скрипт заполняется автоматически, если теги копируются в ручную то требуется в ручную задатать свойство Start Value
   "2080AG505M01.SPSET" : Real AT %DB4151.DBD18, 500 ms
   "2080AG505M01.StatusWork" : Int AT %DB4151.DBW494, 500 ms
   "2080AG505M01.STR01" : Byte AT %DB10.DBB108, 500 ms   // Interlock
   "2080AG505M01.STR01.DefaultText" : TextRef, internal
   "2080AG505M01.STR02" : Byte AT %DB10.DBB109, 500 ms   // Interlock
   "2080AG505M01.STR02.DefaultText" : TextRef, internal
   "2080AG505M01.STR03" : Byte AT %DB10.DBB110, 500 ms   // Interlock
   "2080AG505M01.STR03.DefaultText" : TextRef, internal

HMI tags "2080AG506M01"
   "2080AG506M01.AI1" : Real AT %DB4153.DBD6, 500 ms
   "2080AG506M01.AI2" : Real AT %DB4153.DBD10, 500 ms
   "2080AG506M01.AI3" : Real AT %DB4153.DBD14, 500 ms
   "2080AG506M01.AO1a" : Real AT %DB4153.DBD34, 500 ms
   "2080AG506M01.AO1b" : Real AT %DB4153.DBD38, 500 ms
   "2080AG506M01.AO2a" : Real AT %DB4153.DBD42, 500 ms
   "2080AG506M01.AO2b" : Real AT %DB4153.DBD42, 500 ms
   "2080AG506M01.AO3a" : Real AT %DB4153.DBD50, 500 ms
   "2080AG506M01.AO3b" : Real AT %DB4153.DBD46, 500 ms
   "2080AG506M01.BlockInfo" : Array [0..4] of Int AT %DB4153.DBX74.0, 500 ms
   "2080AG506M01.DefaultText" : TextRef, internal   // Заголовок POPUP окна. При експорте из ECS через скрипт заполняется автоматически, если теги копируются в ручную то требуется в ручную задатать свойство Start Value
   "2080AG506M01.DI.ACK" : Bool AT %DB4153.DBX5.3, 500 ms
   "2080AG506M01.DI.ASTR" : Bool AT %DB4153.DBX2.1, 500 ms
   "2080AG506M01.DI.BUSF" : Bool AT %DB4153.DBX4.5, 500 ms
   "2080AG506M01.DI.DIR" : Bool AT %DB4153.DBX2.2, 500 ms
   "2080AG506M01.DI.DOPR" : Bool AT %DB4153.DBX4.6, 500 ms
   "2080AG506M01.DI.DRDY" : Bool AT %DB4153.DBX3.6, 500 ms
   "2080AG506M01.DI.DTEST" : Bool AT %DB4153.DBX4.7, 500 ms
   "2080AG506M01.DI.EARTH" : Bool AT %DB4153.DBX4.1, 500 ms
   "2080AG506M01.DI.ES" : Bool AT %DB4153.DBX5.2, 500 ms
   "2080AG506M01.DI.GFA" : Bool AT %DB4153.DBX4.3, 500 ms
   "2080AG506M01.DI.GWA" : Bool AT %DB4153.DBX4.4, 500 ms
   "2080AG506M01.DI.LSTP" : Bool AT %DB4153.DBX3.2, 500 ms
   "2080AG506M01.DI.LSTR1" : Bool AT %DB4153.DBX3.0, 500 ms
   "2080AG506M01.DI.LSTR2" : Bool AT %DB4153.DBX3.1, 500 ms
   "2080AG506M01.DI.MCC" : Bool AT %DB4153.DBX2.3, 500 ms
   "2080AG506M01.DI.MD" : Bool AT %DB4153.DBX3.7, 500 ms
   "2080AG506M01.DI.OVL" : Bool AT %DB4153.DBX2.5, 500 ms
   "2080AG506M01.DI.RDY" : Bool AT %DB4153.DBX2.4, 500 ms
   "2080AG506M01.DI.REM" : Bool AT %DB4153.DBX3.3, 500 ms
   "2080AG506M01.DI.RET1" : Bool AT %DB4153.DBX2.6, 500 ms
   "2080AG506M01.DI.RET2" : Bool AT %DB4153.DBX2.7, 500 ms
   "2080AG506M01.DI.SEL" : Bool AT %DB4153.DBX2.0, 500 ms
   "2080AG506M01.DI.SFS" : Bool AT %DB4153.DBX5.0, 500 ms
   "2080AG506M01.DI.SLS" : Bool AT %DB4153.DBX5.1, 500 ms
   "2080AG506M01.DI.SSW" : Bool AT %DB4153.DBX3.4, 500 ms
   "2080AG506M01.DI.STALL" : Bool AT %DB4153.DBX4.0, 500 ms
   "2080AG506M01.DI.TFA" : Bool AT %DB4153.DBX3.5, 500 ms
   "2080AG506M01.DI.UBAL" : Bool AT %DB4153.DBX4.2, 500 ms
   "2080AG506M01.DQ.ASTW" : Bool AT %DB4153.DBX32.0, 500 ms
   "2080AG506M01.DQ.AUT" : Bool AT %DB4153.DBX31.4, 500 ms
   "2080AG506M01.DQ.CON1" : Bool AT %DB4153.DBX30.0, 500 ms
   "2080AG506M01.DQ.CON2" : Bool AT %DB4153.DBX30.1, 500 ms
   "2080AG506M01.DQ.LAMP1" : Bool AT %DB4153.DBX30.2, 500 ms
   "2080AG506M01.DQ.LAMP2" : Bool AT %DB4153.DBX30.3, 500 ms
   "2080AG506M01.DQ.LOC" : Bool AT %DB4153.DBX31.2, 500 ms
   "2080AG506M01.DQ.MAN" : Bool AT %DB4153.DBX31.3, 500 ms
   "2080AG506M01.DQ.OK" : Bool AT %DB4153.DBX31.1, 500 ms
   "2080AG506M01.DQ.RD1" : Bool AT %DB4153.DBX30.5, 500 ms
   "2080AG506M01.DQ.RD2" : Bool AT %DB4153.DBX30.6, 500 ms
   "2080AG506M01.DQ.RES" : Bool AT %DB4153.DBX31.6, 500 ms
   "2080AG506M01.DQ.RUN1" : Bool AT %DB4153.DBX30.7, 500 ms
   "2080AG506M01.DQ.RUN2" : Bool AT %DB4153.DBX31.0, 500 ms
   "2080AG506M01.DQ.SACK" : Bool AT %DB4153.DBX30.4, 500 ms
   "2080AG506M01.DQ.SS" : Bool AT %DB4153.DBX31.5, 500 ms
   "2080AG506M01.DQ.TESTP" : Bool AT %DB4153.DBX31.7, 500 ms
   "2080AG506M01.FP_CMD" : Int AT %DB4153.DBW84, 500 ms
   "2080AG506M01.FP_CMD.AckAlarm" : Bool AT %DB4153.DBX84.7, 500 ms
   "2080AG506M01.FP_CMD.Auto" : Bool AT %DB4153.DBX85.0, 500 ms
   "2080AG506M01.FP_CMD.Local" : Bool AT %DB4153.DBX85.2, 500 ms
   "2080AG506M01.FP_CMD.Manual" : Bool AT %DB4153.DBX85.1, 500 ms
   "2080AG506M01.FP_CMD.QuickStop" : Bool AT %DB4153.DBX84.0, 500 ms
   "2080AG506M01.FP_CMD.Reset" : Bool AT %DB4153.DBX85.6, 500 ms
   "2080AG506M01.FP_CMD.Start1" : Bool AT %DB4153.DBX85.3, 500 ms
   "2080AG506M01.FP_CMD.Start2" : Bool AT %DB4153.DBX85.4, 500 ms
   "2080AG506M01.FP_CMD.Stop" : Bool AT %DB4153.DBX85.5, 500 ms
   "2080AG506M01.FP_CMD.Test" : Bool AT %DB4153.DBX85.7, 500 ms
   "2080AG506M01.FP_DIM.Auto" : Bool AT %DB4153.DBX92.0, 500 ms
   "2080AG506M01.FP_DIM.FP_DIM" : Bool AT %DB4153.DBX92.0, 500 ms
   "2080AG506M01.FP_DIM.Local" : Bool AT %DB4153.DBX92.1, 500 ms
   "2080AG506M01.FP_DIM.Manual" : Bool AT %DB4153.DBX92.2, 500 ms
   "2080AG506M01.FP_DIM.QStop" : Bool AT %DB4153.DBX92.7, 500 ms
   "2080AG506M01.FP_DIM.Reset" : Bool AT %DB4153.DBX93.0, 500 ms
   "2080AG506M01.FP_DIM.Start1" : Bool AT %DB4153.DBX92.3, 500 ms
   "2080AG506M01.FP_DIM.Start2" : Bool AT %DB4153.DBX92.4, 500 ms
   "2080AG506M01.FP_DIM.Stop" : Bool AT %DB4153.DBX92.5, 500 ms
   "2080AG506M01.FP_DIM.TEst" : Bool AT %DB4153.DBX92.6, 500 ms
   "2080AG506M01.FP_DIM1" : Array [0..15] of Bool AT %DB4153.DBX92.0, 500 ms
   "2080AG506M01.FP_EN.Mode_Auto" : Bool AT %DB4153.DBX90.0, 500 ms
   "2080AG506M01.FP_EN.Mode_Loc" : Bool AT %DB4153.DBX90.2, 500 ms
   "2080AG506M01.FP_EN.Mode_Loc_1" : Bool AT %DB4153.DBX90.3, 500 ms
   "2080AG506M01.FP_EN.Mode_Man" : Bool AT %DB4153.DBX90.1, 500 ms
   "2080AG506M01.FP_EN.Mode_SS_Field" : Bool AT %DB4153.DBX90.4, 500 ms
   "2080AG506M01.FP_EN.Mode_SS_FP" : Bool AT %DB4153.DBX90.5, 500 ms
   "2080AG506M01.FP_EN.Mode_Test" : Bool AT %DB4153.DBX90.3, 500 ms
   "2080AG506M01.FP_EN.PB_QStop" : Bool AT %DB4153.DBX90.6, 500 ms
   "2080AG506M01.FP_PARM.AI1_Max" : Real AT %DB4153.DBD158, 500 ms
   "2080AG506M01.FP_PARM.AI1_Min" : Real AT %DB4153.DBD162, 500 ms
   "2080AG506M01.FP_PARM.AI2_Max" : Real AT %DB4153.DBD166, 500 ms
   "2080AG506M01.FP_PARM.AI2_Min" : Real AT %DB4153.DBD170, 500 ms
   "2080AG506M01.FP_PARM.AI3_Max" : Real AT %DB4153.DBD174, 500 ms
   "2080AG506M01.FP_PARM.AI3_Min" : Real AT %DB4153.DBD178, 500 ms
   "2080AG506M01.FP_PARM.AO1a_Max" : Real AT %DB4153.DBD182, 500 ms
   "2080AG506M01.FP_PARM.AO1a_Min" : Real AT %DB4153.DBD186, 500 ms
   "2080AG506M01.FP_PARM.AO1b_Max" : Real AT %DB4153.DBD206, 500 ms
   "2080AG506M01.FP_PARM.AO1b_Min" : Real AT %DB4153.DBD210, 500 ms
   "2080AG506M01.FP_PARM.AO2a_Max" : Real AT %DB4153.DBD190, 500 ms
   "2080AG506M01.FP_PARM.AO2a_Min" : Real AT %DB4153.DBD194, 500 ms
   "2080AG506M01.FP_PARM.AO2b_Max" : Real AT %DB4153.DBD214, 500 ms
   "2080AG506M01.FP_PARM.AO2b_Min" : Real AT %DB4153.DBD218, 500 ms
   "2080AG506M01.FP_PARM.AO3a_Max" : Real AT %DB4153.DBD198, 500 ms
   "2080AG506M01.FP_PARM.AO3a_Min" : Real AT %DB4153.DBD202, 500 ms
   "2080AG506M01.FP_PARM.AO3b_Max" : Real AT %DB4153.DBD222, 500 ms
   "2080AG506M01.FP_PARM.AO3b_Min" : Real AT %DB4153.DBD226, 500 ms
   "2080AG506M01.FP_PARM.ChangeDir_Acc" : Int AT %DB4153.DBW138, 500 ms
   "2080AG506M01.FP_PARM.ChangeDir_Pre" : Int AT %DB4153.DBW136, 500 ms
   "2080AG506M01.FP_PARM.DelayStart_Acc" : Int AT %DB4153.DBW114, 500 ms
   "2080AG506M01.FP_PARM.DelayStart_Pre" : Int AT %DB4153.DBW112, 500 ms
   "2080AG506M01.FP_PARM.DelayStop_Acc" : Int AT %DB4153.DBW118, 500 ms
   "2080AG506M01.FP_PARM.DelayStop_Pre" : Int AT %DB4153.DBW116, 500 ms
   "2080AG506M01.FP_PARM.INTL" : Bool AT %DB4153.DBX230.0, 500 ms
   "2080AG506M01.FP_PARM.INTL_SEQ_STP" : Bool AT %DB4153.DBX230.3, 500 ms
   "2080AG506M01.FP_PARM.INTL_SEQ_STR1" : Bool AT %DB4153.DBX230.1, 500 ms
   "2080AG506M01.FP_PARM.INTL_SEQ_STR2" : Bool AT %DB4153.DBX230.2, 500 ms
   "2080AG506M01.FP_PARM.LeaveFS_Acc" : Int AT %DB4153.DBW142, 500 ms
   "2080AG506M01.FP_PARM.LeaveFS_Pre" : Int AT %DB4153.DBW140, 500 ms
   "2080AG506M01.FP_PARM.MD_Freq_PV" : Int AT %DB4153.DBW154, 500 ms
   "2080AG506M01.FP_PARM.MD_Freq_SP" : Int AT %DB4153.DBW152, 500 ms
   "2080AG506M01.FP_PARM.ReachFS_Acc" : Int AT %DB4153.DBW150, 500 ms
   "2080AG506M01.FP_PARM.ReachFS_Pre" : Int AT %DB4153.DBW148, 500 ms
   "2080AG506M01.FP_PARM.ReachLS_Acc" : Int AT %DB4153.DBW146, 500 ms
   "2080AG506M01.FP_PARM.ReachLS_Pre" : Int AT %DB4153.DBW144, 500 ms
   "2080AG506M01.FP_PARM.ReturnMon_Acc" : Int AT %DB4153.DBW122, 500 ms
   "2080AG506M01.FP_PARM.ReturnMon_Pre" : Int AT %DB4153.DBW120, 500 ms
   "2080AG506M01.FP_PARM.RunDelay1_Acc" : Int AT %DB4153.DBW106, 500 ms
   "2080AG506M01.FP_PARM.RunDelay1_Pre" : Int AT %DB4153.DBW104, 500 ms
   "2080AG506M01.FP_PARM.RunDelay2_Acc" : Int AT %DB4153.DBW110, 500 ms
   "2080AG506M01.FP_PARM.RunDelay2_Pre" : Int AT %DB4153.DBW108, 500 ms
   "2080AG506M01.FP_PARM.SpeedMonOffDelay_Acc" : Int AT %DB4153.DBW130, 500 ms
   "2080AG506M01.FP_PARM.SpeedMonOffDelay_Pre" : Int AT %DB4153.DBW128, 500 ms
   "2080AG506M01.FP_PARM.SpeedMonOnDelay_Acc" : Int AT %DB4153.DBW126, 500 ms
   "2080AG506M01.FP_PARM.SpeedMonOnDelay_Pre" : Int AT %DB4153.DBW124, 500 ms
   "2080AG506M01.FP_PARM.SpeedMonTrigDelay_Acc" : Int AT %DB4153.DBW134, 500 ms
   "2080AG506M01.FP_PARM.SpeedMonTrigDelay_Pre" : Int AT %DB4153.DBW132, 500 ms
   "2080AG506M01.FP_PARM.StartWarn_Acc" : Int AT %DB4153.DBW102, 500 ms
   "2080AG506M01.FP_PARM.StartWarn_Pre" : Int AT %DB4153.DBW100, 500 ms
   "2080AG506M01.FP_PARM.StopReason" : Int AT %DB4153.DBW156, 500 ms
   "2080AG506M01.FP_SEL.INCH_Loc" : Bool AT %DB4153.DBX87.7, 500 ms
   "2080AG506M01.FP_SEL.INCH_Man" : Bool AT %DB4153.DBX87.6, 500 ms
   "2080AG506M01.FP_SEL.MD" : Bool AT %DB4153.DBX86.0, 500 ms
   "2080AG506M01.FP_SEL.MD_Maintain" : Bool AT %DB4153.DBX86.3, 500 ms
   "2080AG506M01.FP_SEL.MD_OnOff" : Bool AT %DB4153.DBX86.2, 500 ms
   "2080AG506M01.FP_SEL.MD_Puls" : Bool AT %DB4153.DBX86.1, 500 ms
   "2080AG506M01.FP_SEL.MotorStarter" : Bool AT %DB4153.DBX87.3, 500 ms
   "2080AG506M01.FP_SEL.OutOfSevice" : Bool AT %DB4153.DBX88.0, 500 ms
   "2080AG506M01.FP_SEL.ParentCollection" : Bool AT %DB4153.DBX87.5, 500 ms
   "2080AG506M01.FP_SEL.ParentSupress" : Bool AT %DB4153.DBX87.4, 500 ms
   "2080AG506M01.FP_SEL.STW_AutoStart" : Bool AT %DB4153.DBX86.4, 500 ms
   "2080AG506M01.FP_SEL.STW_Local" : Bool AT %DB4153.DBX86.5, 500 ms
   "2080AG506M01.FP_SEL.STW_Manual" : Bool AT %DB4153.DBX86.6, 500 ms
   "2080AG506M01.FP_SEL.STW_Single" : Bool AT %DB4153.DBX86.7, 500 ms
   "2080AG506M01.FP_SEL.Type_Bimotor" : Bool AT %DB4153.DBX87.1, 500 ms
   "2080AG506M01.FP_SEL.Type_Indication" : Bool AT %DB4153.DBX87.2, 500 ms
   "2080AG506M01.FP_SEL.Type_Unimotor" : Bool AT %DB4153.DBX87.0, 500 ms
   "2080AG506M01.FP_SEL.WarningDrive" : Bool AT %DB4153.DBX88.1, 500 ms
   "2080AG506M01.FP_SHOW.ACK" : Bool AT %DB4153.DBX97.5, 500 ms
   "2080AG506M01.FP_SHOW.AI1" : Bool AT %DB4153.DBX95.0, 500 ms
   "2080AG506M01.FP_SHOW.AI2" : Bool AT %DB4153.DBX95.1, 500 ms
   "2080AG506M01.FP_SHOW.AI3" : Bool AT %DB4153.DBX95.2, 500 ms
   "2080AG506M01.FP_SHOW.ASTR" : Bool AT %DB4153.DBX99.2, 500 ms
   "2080AG506M01.FP_SHOW.B1" : Byte AT %DB4153.DBB95, 500 ms
   "2080AG506M01.FP_SHOW.B2" : Byte AT %DB4153.DBB96, 500 ms
   "2080AG506M01.FP_SHOW.B3" : Byte AT %DB4153.DBB97, 500 ms
   "2080AG506M01.FP_SHOW.B4" : Byte AT %DB4153.DBB98, 500 ms
   "2080AG506M01.FP_SHOW.BUSF" : Bool AT %DB4153.DBX97.2, 500 ms
   "2080AG506M01.FP_SHOW.ChangeDir" : Bool AT %DB4153.DBX99.0, 500 ms
   "2080AG506M01.FP_SHOW.CON2" : Bool AT %DB4153.DBX98.2, 500 ms
   "2080AG506M01.FP_SHOW.DelayRun2" : Bool AT %DB4153.DBX98.7, 500 ms
   "2080AG506M01.FP_SHOW.DOPR" : Bool AT %DB4153.DBX97.3, 500 ms
   "2080AG506M01.FP_SHOW.DRDY" : Bool AT %DB4153.DBX96.4, 500 ms
   "2080AG506M01.FP_SHOW.DTEST" : Bool AT %DB4153.DBX97.4, 500 ms
   "2080AG506M01.FP_SHOW.EARTH" : Bool AT %DB4153.DBX96.6, 500 ms
   "2080AG506M01.FP_SHOW.ES" : Bool AT %DB4153.DBX96.2, 500 ms
   "2080AG506M01.FP_SHOW.GFA" : Bool AT %DB4153.DBX97.0, 500 ms
   "2080AG506M01.FP_SHOW.GWA" : Bool AT %DB4153.DBX97.1, 500 ms
   "2080AG506M01.FP_SHOW.LSTP" : Bool AT %DB4153.DBX95.7, 500 ms
   "2080AG506M01.FP_SHOW.LSTR1" : Bool AT %DB4153.DBX97.6, 500 ms
   "2080AG506M01.FP_SHOW.LSTR2" : Bool AT %DB4153.DBX97.7, 500 ms
   "2080AG506M01.FP_SHOW.MCC" : Bool AT %DB4153.DBX95.4, 500 ms
   "2080AG506M01.FP_SHOW.MD" : Bool AT %DB4153.DBX98.6, 500 ms
   "2080AG506M01.FP_SHOW.OVL" : Bool AT %DB4153.DBX95.6, 500 ms
   "2080AG506M01.FP_SHOW.PB_Auto" : Bool AT %DB4153.DBX94.0, 500 ms
   "2080AG506M01.FP_SHOW.PB_Local" : Bool AT %DB4153.DBX94.1, 500 ms
   "2080AG506M01.FP_SHOW.PB_Manual" : Bool AT %DB4153.DBX94.2, 500 ms
   "2080AG506M01.FP_SHOW.PB_QStop" : Bool AT %DB4153.DBX94.7, 500 ms
   "2080AG506M01.FP_SHOW.PB_Reset" : Bool AT %DB4153.DBX99.1, 500 ms
   "2080AG506M01.FP_SHOW.PB_Start1" : Bool AT %DB4153.DBX94.3, 500 ms
   "2080AG506M01.FP_SHOW.PB_Start2" : Bool AT %DB4153.DBX94.4, 500 ms
   "2080AG506M01.FP_SHOW.PB_Stop" : Bool AT %DB4153.DBX94.5, 500 ms
   "2080AG506M01.FP_SHOW.PB_Test" : Bool AT %DB4153.DBX94.6, 500 ms
   "2080AG506M01.FP_SHOW.RD2" : Bool AT %DB4153.DBX98.3, 500 ms
   "2080AG506M01.FP_SHOW.RDY" : Bool AT %DB4153.DBX95.5, 500 ms
   "2080AG506M01.FP_SHOW.REM" : Bool AT %DB4153.DBX96.0, 500 ms
   "2080AG506M01.FP_SHOW.RET2" : Bool AT %DB4153.DBX98.0, 500 ms
   "2080AG506M01.FP_SHOW.RUN2" : Bool AT %DB4153.DBX98.1, 500 ms
   "2080AG506M01.FP_SHOW.SFS" : Bool AT %DB4153.DBX98.4, 500 ms
   "2080AG506M01.FP_SHOW.SLS" : Bool AT %DB4153.DBX98.5, 500 ms
   "2080AG506M01.FP_SHOW.SP" : Bool AT %DB4153.DBX95.3, 500 ms
   "2080AG506M01.FP_SHOW.SSW" : Bool AT %DB4153.DBX96.1, 500 ms
   "2080AG506M01.FP_SHOW.STALL" : Bool AT %DB4153.DBX96.5, 500 ms
   "2080AG506M01.FP_SHOW.TFA" : Bool AT %DB4153.DBX96.3, 500 ms
   "2080AG506M01.FP_SHOW.UBAL" : Bool AT %DB4153.DBX96.7, 500 ms
   "2080AG506M01.ModePointer" : Int AT %DB4153.DBW496, 500 ms
   "2080AG506M01.MSW" : DWord AT %DB4153.DBD62, 500 ms
   "2080AG506M01.ParentInfo" : TextRef, internal   // Имя родителя для попап окна, вкладка инфо. При експорте из ECS через скрипт заполняется автоматически, если теги копируются в ручную то требуется в ручную задатать свойство Start Value
   "2080AG506M01.SPSET" : Real AT %DB4153.DBD18, 500 ms
   "2080AG506M01.StatusWork" : Int AT %DB4153.DBW494, 500 ms
   "2080AG506M01.STR01" : Byte AT %DB10.DBB112, 500 ms   // Interlock
   "2080AG506M01.STR01.DefaultText" : TextRef, internal
   "2080AG506M01.STR02" : Byte AT %DB10.DBB113, 500 ms   // Interlock
   "2080AG506M01.STR02.DefaultText" : TextRef, internal

HMI tags "2080AG507M01"
   "2080AG507M01.AI1" : Real AT %DB4155.DBD6, 500 ms
   "2080AG507M01.AI2" : Real AT %DB4155.DBD10, 500 ms
   "2080AG507M01.AI3" : Real AT %DB4155.DBD14, 500 ms
   "2080AG507M01.AO1a" : Real AT %DB4155.DBD34, 500 ms
   "2080AG507M01.AO1b" : Real AT %DB4155.DBD38, 500 ms
   "2080AG507M01.AO2a" : Real AT %DB4155.DBD42, 500 ms
   "2080AG507M01.AO2b" : Real AT %DB4155.DBD42, 500 ms
   "2080AG507M01.AO3a" : Real AT %DB4155.DBD50, 500 ms
   "2080AG507M01.AO3b" : Real AT %DB4155.DBD46, 500 ms
   "2080AG507M01.BlockInfo" : Array [0..4] of Int AT %DB4155.DBX74.0, 500 ms
   "2080AG507M01.DefaultText" : TextRef, internal   // Заголовок POPUP окна. При експорте из ECS через скрипт заполняется автоматически, если теги копируются в ручную то требуется в ручную задатать свойство Start Value
   "2080AG507M01.DI.ACK" : Bool AT %DB4155.DBX5.3, 500 ms
   "2080AG507M01.DI.ASTR" : Bool AT %DB4155.DBX2.1, 500 ms
   "2080AG507M01.DI.BUSF" : Bool AT %DB4155.DBX4.5, 500 ms
   "2080AG507M01.DI.DIR" : Bool AT %DB4155.DBX2.2, 500 ms
   "2080AG507M01.DI.DOPR" : Bool AT %DB4155.DBX4.6, 500 ms
   "2080AG507M01.DI.DRDY" : Bool AT %DB4155.DBX3.6, 500 ms
   "2080AG507M01.DI.DTEST" : Bool AT %DB4155.DBX4.7, 500 ms
   "2080AG507M01.DI.EARTH" : Bool AT %DB4155.DBX4.1, 500 ms
   "2080AG507M01.DI.ES" : Bool AT %DB4155.DBX5.2, 500 ms
   "2080AG507M01.DI.GFA" : Bool AT %DB4155.DBX4.3, 500 ms
   "2080AG507M01.DI.GWA" : Bool AT %DB4155.DBX4.4, 500 ms
   "2080AG507M01.DI.LSTP" : Bool AT %DB4155.DBX3.2, 500 ms
   "2080AG507M01.DI.LSTR1" : Bool AT %DB4155.DBX3.0, 500 ms
   "2080AG507M01.DI.LSTR2" : Bool AT %DB4155.DBX3.1, 500 ms
   "2080AG507M01.DI.MCC" : Bool AT %DB4155.DBX2.3, 500 ms
   "2080AG507M01.DI.MD" : Bool AT %DB4155.DBX3.7, 500 ms
   "2080AG507M01.DI.OVL" : Bool AT %DB4155.DBX2.5, 500 ms
   "2080AG507M01.DI.RDY" : Bool AT %DB4155.DBX2.4, 500 ms
   "2080AG507M01.DI.REM" : Bool AT %DB4155.DBX3.3, 500 ms
   "2080AG507M01.DI.RET1" : Bool AT %DB4155.DBX2.6, 500 ms
   "2080AG507M01.DI.RET2" : Bool AT %DB4155.DBX2.7, 500 ms
   "2080AG507M01.DI.SEL" : Bool AT %DB4155.DBX2.0, 500 ms
   "2080AG507M01.DI.SFS" : Bool AT %DB4155.DBX5.0, 500 ms
   "2080AG507M01.DI.SLS" : Bool AT %DB4155.DBX5.1, 500 ms
   "2080AG507M01.DI.SSW" : Bool AT %DB4155.DBX3.4, 500 ms
   "2080AG507M01.DI.STALL" : Bool AT %DB4155.DBX4.0, 500 ms
   "2080AG507M01.DI.TFA" : Bool AT %DB4155.DBX3.5, 500 ms
   "2080AG507M01.DI.UBAL" : Bool AT %DB4155.DBX4.2, 500 ms
   "2080AG507M01.DQ.ASTW" : Bool AT %DB4155.DBX32.0, 500 ms
   "2080AG507M01.DQ.AUT" : Bool AT %DB4155.DBX31.4, 500 ms
   "2080AG507M01.DQ.CON1" : Bool AT %DB4155.DBX30.0, 500 ms
   "2080AG507M01.DQ.CON2" : Bool AT %DB4155.DBX30.1, 500 ms
   "2080AG507M01.DQ.LAMP1" : Bool AT %DB4155.DBX30.2, 500 ms
   "2080AG507M01.DQ.LAMP2" : Bool AT %DB4155.DBX30.3, 500 ms
   "2080AG507M01.DQ.LOC" : Bool AT %DB4155.DBX31.2, 500 ms
   "2080AG507M01.DQ.MAN" : Bool AT %DB4155.DBX31.3, 500 ms
   "2080AG507M01.DQ.OK" : Bool AT %DB4155.DBX31.1, 500 ms
   "2080AG507M01.DQ.RD1" : Bool AT %DB4155.DBX30.5, 500 ms
   "2080AG507M01.DQ.RD2" : Bool AT %DB4155.DBX30.6, 500 ms
   "2080AG507M01.DQ.RES" : Bool AT %DB4155.DBX31.6, 500 ms
   "2080AG507M01.DQ.RUN1" : Bool AT %DB4155.DBX30.7, 500 ms
   "2080AG507M01.DQ.RUN2" : Bool AT %DB4155.DBX31.0, 500 ms
   "2080AG507M01.DQ.SACK" : Bool AT %DB4155.DBX30.4, 500 ms
   "2080AG507M01.DQ.SS" : Bool AT %DB4155.DBX31.5, 500 ms
   "2080AG507M01.DQ.TESTP" : Bool AT %DB4155.DBX31.7, 500 ms
   "2080AG507M01.FP_CMD" : Int AT %DB4155.DBW84, 500 ms
   "2080AG507M01.FP_CMD.AckAlarm" : Bool AT %DB4155.DBX84.7, 500 ms
   "2080AG507M01.FP_CMD.Auto" : Bool AT %DB4155.DBX85.0, 500 ms
   "2080AG507M01.FP_CMD.Local" : Bool AT %DB4155.DBX85.2, 500 ms
   "2080AG507M01.FP_CMD.Manual" : Bool AT %DB4155.DBX85.1, 500 ms
   "2080AG507M01.FP_CMD.QuickStop" : Bool AT %DB4155.DBX84.0, 500 ms
   "2080AG507M01.FP_CMD.Reset" : Bool AT %DB4155.DBX85.6, 500 ms
   "2080AG507M01.FP_CMD.Start1" : Bool AT %DB4155.DBX85.3, 500 ms
   "2080AG507M01.FP_CMD.Start2" : Bool AT %DB4155.DBX85.4, 500 ms
   "2080AG507M01.FP_CMD.Stop" : Bool AT %DB4155.DBX85.5, 500 ms
   "2080AG507M01.FP_CMD.Test" : Bool AT %DB4155.DBX85.7, 500 ms
   "2080AG507M01.FP_DIM.Auto" : Bool AT %DB4155.DBX92.0, 500 ms
   "2080AG507M01.FP_DIM.FP_DIM" : Bool AT %DB4155.DBX92.0, 500 ms
   "2080AG507M01.FP_DIM.Local" : Bool AT %DB4155.DBX92.1, 500 ms
   "2080AG507M01.FP_DIM.Manual" : Bool AT %DB4155.DBX92.2, 500 ms
   "2080AG507M01.FP_DIM.QStop" : Bool AT %DB4155.DBX92.7, 500 ms
   "2080AG507M01.FP_DIM.Reset" : Bool AT %DB4155.DBX93.0, 500 ms
   "2080AG507M01.FP_DIM.Start1" : Bool AT %DB4155.DBX92.3, 500 ms
   "2080AG507M01.FP_DIM.Start2" : Bool AT %DB4155.DBX92.4, 500 ms
   "2080AG507M01.FP_DIM.Stop" : Bool AT %DB4155.DBX92.5, 500 ms
   "2080AG507M01.FP_DIM.TEst" : Bool AT %DB4155.DBX92.6, 500 ms
   "2080AG507M01.FP_DIM1" : Array [0..15] of Bool AT %DB4155.DBX92.0, 500 ms
   "2080AG507M01.FP_EN.Mode_Auto" : Bool AT %DB4155.DBX90.0, 500 ms
   "2080AG507M01.FP_EN.Mode_Loc" : Bool AT %DB4155.DBX90.2, 500 ms
   "2080AG507M01.FP_EN.Mode_Loc_1" : Bool AT %DB4155.DBX90.3, 500 ms
   "2080AG507M01.FP_EN.Mode_Man" : Bool AT %DB4155.DBX90.1, 500 ms
   "2080AG507M01.FP_EN.Mode_SS_Field" : Bool AT %DB4155.DBX90.4, 500 ms
   "2080AG507M01.FP_EN.Mode_SS_FP" : Bool AT %DB4155.DBX90.5, 500 ms
   "2080AG507M01.FP_EN.Mode_Test" : Bool AT %DB4155.DBX90.3, 500 ms
   "2080AG507M01.FP_EN.PB_QStop" : Bool AT %DB4155.DBX90.6, 500 ms
   "2080AG507M01.FP_PARM.AI1_Max" : Real AT %DB4155.DBD158, 500 ms
   "2080AG507M01.FP_PARM.AI1_Min" : Real AT %DB4155.DBD162, 500 ms
   "2080AG507M01.FP_PARM.AI2_Max" : Real AT %DB4155.DBD166, 500 ms
   "2080AG507M01.FP_PARM.AI2_Min" : Real AT %DB4155.DBD170, 500 ms
   "2080AG507M01.FP_PARM.AI3_Max" : Real AT %DB4155.DBD174, 500 ms
   "2080AG507M01.FP_PARM.AI3_Min" : Real AT %DB4155.DBD178, 500 ms
   "2080AG507M01.FP_PARM.AO1a_Max" : Real AT %DB4155.DBD182, 500 ms
   "2080AG507M01.FP_PARM.AO1a_Min" : Real AT %DB4155.DBD186, 500 ms
   "2080AG507M01.FP_PARM.AO1b_Max" : Real AT %DB4155.DBD206, 500 ms
   "2080AG507M01.FP_PARM.AO1b_Min" : Real AT %DB4155.DBD210, 500 ms
   "2080AG507M01.FP_PARM.AO2a_Max" : Real AT %DB4155.DBD190, 500 ms
   "2080AG507M01.FP_PARM.AO2a_Min" : Real AT %DB4155.DBD194, 500 ms
   "2080AG507M01.FP_PARM.AO2b_Max" : Real AT %DB4155.DBD214, 500 ms
   "2080AG507M01.FP_PARM.AO2b_Min" : Real AT %DB4155.DBD218, 500 ms
   "2080AG507M01.FP_PARM.AO3a_Max" : Real AT %DB4155.DBD198, 500 ms
   "2080AG507M01.FP_PARM.AO3a_Min" : Real AT %DB4155.DBD202, 500 ms
   "2080AG507M01.FP_PARM.AO3b_Max" : Real AT %DB4155.DBD222, 500 ms
   "2080AG507M01.FP_PARM.AO3b_Min" : Real AT %DB4155.DBD226, 500 ms
   "2080AG507M01.FP_PARM.ChangeDir_Acc" : Int AT %DB4155.DBW138, 500 ms
   "2080AG507M01.FP_PARM.ChangeDir_Pre" : Int AT %DB4155.DBW136, 500 ms
   "2080AG507M01.FP_PARM.DelayStart_Acc" : Int AT %DB4155.DBW114, 500 ms
   "2080AG507M01.FP_PARM.DelayStart_Pre" : Int AT %DB4155.DBW112, 500 ms
   "2080AG507M01.FP_PARM.DelayStop_Acc" : Int AT %DB4155.DBW118, 500 ms
   "2080AG507M01.FP_PARM.DelayStop_Pre" : Int AT %DB4155.DBW116, 500 ms
   "2080AG507M01.FP_PARM.INTL" : Bool AT %DB4155.DBX230.0, 500 ms
   "2080AG507M01.FP_PARM.INTL_SEQ_STP" : Bool AT %DB4155.DBX230.3, 500 ms
   "2080AG507M01.FP_PARM.INTL_SEQ_STR1" : Bool AT %DB4155.DBX230.1, 500 ms
   "2080AG507M01.FP_PARM.INTL_SEQ_STR2" : Bool AT %DB4155.DBX230.2, 500 ms
   "2080AG507M01.FP_PARM.LeaveFS_Acc" : Int AT %DB4155.DBW142, 500 ms
   "2080AG507M01.FP_PARM.LeaveFS_Pre" : Int AT %DB4155.DBW140, 500 ms
   "2080AG507M01.FP_PARM.MD_Freq_PV" : Int AT %DB4155.DBW154, 500 ms
   "2080AG507M01.FP_PARM.MD_Freq_SP" : Int AT %DB4155.DBW152, 500 ms
   "2080AG507M01.FP_PARM.ReachFS_Acc" : Int AT %DB4155.DBW150, 500 ms
   "2080AG507M01.FP_PARM.ReachFS_Pre" : Int AT %DB4155.DBW148, 500 ms
   "2080AG507M01.FP_PARM.ReachLS_Acc" : Int AT %DB4155.DBW146, 500 ms
   "2080AG507M01.FP_PARM.ReachLS_Pre" : Int AT %DB4155.DBW144, 500 ms
   "2080AG507M01.FP_PARM.ReturnMon_Acc" : Int AT %DB4155.DBW122, 500 ms
   "2080AG507M01.FP_PARM.ReturnMon_Pre" : Int AT %DB4155.DBW120, 500 ms
   "2080AG507M01.FP_PARM.RunDelay1_Acc" : Int AT %DB4155.DBW106, 500 ms
   "2080AG507M01.FP_PARM.RunDelay1_Pre" : Int AT %DB4155.DBW104, 500 ms
   "2080AG507M01.FP_PARM.RunDelay2_Acc" : Int AT %DB4155.DBW110, 500 ms
   "2080AG507M01.FP_PARM.RunDelay2_Pre" : Int AT %DB4155.DBW108, 500 ms
   "2080AG507M01.FP_PARM.SpeedMonOffDelay_Acc" : Int AT %DB4155.DBW130, 500 ms
   "2080AG507M01.FP_PARM.SpeedMonOffDelay_Pre" : Int AT %DB4155.DBW128, 500 ms
   "2080AG507M01.FP_PARM.SpeedMonOnDelay_Acc" : Int AT %DB4155.DBW126, 500 ms
   "2080AG507M01.FP_PARM.SpeedMonOnDelay_Pre" : Int AT %DB4155.DBW124, 500 ms
   "2080AG507M01.FP_PARM.SpeedMonTrigDelay_Acc" : Int AT %DB4155.DBW134, 500 ms
   "2080AG507M01.FP_PARM.SpeedMonTrigDelay_Pre" : Int AT %DB4155.DBW132, 500 ms
   "2080AG507M01.FP_PARM.StartWarn_Acc" : Int AT %DB4155.DBW102, 500 ms
   "2080AG507M01.FP_PARM.StartWarn_Pre" : Int AT %DB4155.DBW100, 500 ms
   "2080AG507M01.FP_PARM.StopReason" : Int AT %DB4155.DBW156, 500 ms
   "2080AG507M01.FP_SEL.INCH_Loc" : Bool AT %DB4155.DBX87.7, 500 ms
   "2080AG507M01.FP_SEL.INCH_Man" : Bool AT %DB4155.DBX87.6, 500 ms
   "2080AG507M01.FP_SEL.MD" : Bool AT %DB4155.DBX86.0, 500 ms
   "2080AG507M01.FP_SEL.MD_Maintain" : Bool AT %DB4155.DBX86.3, 500 ms
   "2080AG507M01.FP_SEL.MD_OnOff" : Bool AT %DB4155.DBX86.2, 500 ms
   "2080AG507M01.FP_SEL.MD_Puls" : Bool AT %DB4155.DBX86.1, 500 ms
   "2080AG507M01.FP_SEL.MotorStarter" : Bool AT %DB4155.DBX87.3, 500 ms
   "2080AG507M01.FP_SEL.OutOfSevice" : Bool AT %DB4155.DBX88.0, 500 ms
   "2080AG507M01.FP_SEL.ParentCollection" : Bool AT %DB4155.DBX87.5, 500 ms
   "2080AG507M01.FP_SEL.ParentSupress" : Bool AT %DB4155.DBX87.4, 500 ms
   "2080AG507M01.FP_SEL.STW_AutoStart" : Bool AT %DB4155.DBX86.4, 500 ms
   "2080AG507M01.FP_SEL.STW_Local" : Bool AT %DB4155.DBX86.5, 500 ms
   "2080AG507M01.FP_SEL.STW_Manual" : Bool AT %DB4155.DBX86.6, 500 ms
   "2080AG507M01.FP_SEL.STW_Single" : Bool AT %DB4155.DBX86.7, 500 ms
   "2080AG507M01.FP_SEL.Type_Bimotor" : Bool AT %DB4155.DBX87.1, 500 ms
   "2080AG507M01.FP_SEL.Type_Indication" : Bool AT %DB4155.DBX87.2, 500 ms
   "2080AG507M01.FP_SEL.Type_Unimotor" : Bool AT %DB4155.DBX87.0, 500 ms
   "2080AG507M01.FP_SEL.WarningDrive" : Bool AT %DB4155.DBX88.1, 500 ms
   "2080AG507M01.FP_SHOW.ACK" : Bool AT %DB4155.DBX97.5, 500 ms
   "2080AG507M01.FP_SHOW.AI1" : Bool AT %DB4155.DBX95.0, 500 ms
   "2080AG507M01.FP_SHOW.AI2" : Bool AT %DB4155.DBX95.1, 500 ms
   "2080AG507M01.FP_SHOW.AI3" : Bool AT %DB4155.DBX95.2, 500 ms
   "2080AG507M01.FP_SHOW.ASTR" : Bool AT %DB4155.DBX99.2, 500 ms
   "2080AG507M01.FP_SHOW.B1" : Byte AT %DB4155.DBB95, 500 ms
   "2080AG507M01.FP_SHOW.B2" : Byte AT %DB4155.DBB96, 500 ms
   "2080AG507M01.FP_SHOW.B3" : Byte AT %DB4155.DBB97, 500 ms
   "2080AG507M01.FP_SHOW.B4" : Byte AT %DB4155.DBB98, 500 ms
   "2080AG507M01.FP_SHOW.BUSF" : Bool AT %DB4155.DBX97.2, 500 ms
   "2080AG507M01.FP_SHOW.ChangeDir" : Bool AT %DB4155.DBX99.0, 500 ms
   "2080AG507M01.FP_SHOW.CON2" : Bool AT %DB4155.DBX98.2, 500 ms
   "2080AG507M01.FP_SHOW.DelayRun2" : Bool AT %DB4155.DBX98.7, 500 ms
   "2080AG507M01.FP_SHOW.DOPR" : Bool AT %DB4155.DBX97.3, 500 ms
   "2080AG507M01.FP_SHOW.DRDY" : Bool AT %DB4155.DBX96.4, 500 ms
   "2080AG507M01.FP_SHOW.DTEST" : Bool AT %DB4155.DBX97.4, 500 ms
   "2080AG507M01.FP_SHOW.EARTH" : Bool AT %DB4155.DBX96.6, 500 ms
   "2080AG507M01.FP_SHOW.ES" : Bool AT %DB4155.DBX96.2, 500 ms
   "2080AG507M01.FP_SHOW.GFA" : Bool AT %DB4155.DBX97.0, 500 ms
   "2080AG507M01.FP_SHOW.GWA" : Bool AT %DB4155.DBX97.1, 500 ms
   "2080AG507M01.FP_SHOW.LSTP" : Bool AT %DB4155.DBX95.7, 500 ms
   "2080AG507M01.FP_SHOW.LSTR1" : Bool AT %DB4155.DBX97.6, 500 ms
   "2080AG507M01.FP_SHOW.LSTR2" : Bool AT %DB4155.DBX97.7, 500 ms
   "2080AG507M01.FP_SHOW.MCC" : Bool AT %DB4155.DBX95.4, 500 ms
   "2080AG507M01.FP_SHOW.MD" : Bool AT %DB4155.DBX98.6, 500 ms
   "2080AG507M01.FP_SHOW.OVL" : Bool AT %DB4155.DBX95.6, 500 ms
   "2080AG507M01.FP_SHOW.PB_Auto" : Bool AT %DB4155.DBX94.0, 500 ms
   "2080AG507M01.FP_SHOW.PB_Local" : Bool AT %DB4155.DBX94.1, 500 ms
   "2080AG507M01.FP_SHOW.PB_Manual" : Bool AT %DB4155.DBX94.2, 500 ms
   "2080AG507M01.FP_SHOW.PB_QStop" : Bool AT %DB4155.DBX94.7, 500 ms
   "2080AG507M01.FP_SHOW.PB_Reset" : Bool AT %DB4155.DBX99.1, 500 ms
   "2080AG507M01.FP_SHOW.PB_Start1" : Bool AT %DB4155.DBX94.3, 500 ms
   "2080AG507M01.FP_SHOW.PB_Start2" : Bool AT %DB4155.DBX94.4, 500 ms
   "2080AG507M01.FP_SHOW.PB_Stop" : Bool AT %DB4155.DBX94.5, 500 ms
   "2080AG507M01.FP_SHOW.PB_Test" : Bool AT %DB4155.DBX94.6, 500 ms
   "2080AG507M01.FP_SHOW.RD2" : Bool AT %DB4155.DBX98.3, 500 ms
   "2080AG507M01.FP_SHOW.RDY" : Bool AT %DB4155.DBX95.5, 500 ms
   "2080AG507M01.FP_SHOW.REM" : Bool AT %DB4155.DBX96.0, 500 ms
   "2080AG507M01.FP_SHOW.RET2" : Bool AT %DB4155.DBX98.0, 500 ms
   "2080AG507M01.FP_SHOW.RUN2" : Bool AT %DB4155.DBX98.1, 500 ms
   "2080AG507M01.FP_SHOW.SFS" : Bool AT %DB4155.DBX98.4, 500 ms
   "2080AG507M01.FP_SHOW.SLS" : Bool AT %DB4155.DBX98.5, 500 ms
   "2080AG507M01.FP_SHOW.SP" : Bool AT %DB4155.DBX95.3, 500 ms
   "2080AG507M01.FP_SHOW.SSW" : Bool AT %DB4155.DBX96.1, 500 ms
   "2080AG507M01.FP_SHOW.STALL" : Bool AT %DB4155.DBX96.5, 500 ms
   "2080AG507M01.FP_SHOW.TFA" : Bool AT %DB4155.DBX96.3, 500 ms
   "2080AG507M01.FP_SHOW.UBAL" : Bool AT %DB4155.DBX96.7, 500 ms
   "2080AG507M01.ModePointer" : Int AT %DB4155.DBW496, 500 ms
   "2080AG507M01.MSW" : DWord AT %DB4155.DBD62, 500 ms
   "2080AG507M01.ParentInfo" : TextRef, internal   // Имя родителя для попап окна, вкладка инфо. При експорте из ECS через скрипт заполняется автоматически, если теги копируются в ручную то требуется в ручную задатать свойство Start Value
   "2080AG507M01.SPSET" : Real AT %DB4155.DBD18, 500 ms
   "2080AG507M01.StatusWork" : Int AT %DB4155.DBW494, 500 ms
   "2080AG507M01.STR01" : Byte AT %DB10.DBB115, 500 ms   // Interlock
   "2080AG507M01.STR01.DefaultText" : TextRef, internal

HMI tags "2080AG508M01"
   "2080AG508M01.AI1" : Real AT %DB4300.DBD6, 500 ms
   "2080AG508M01.AI2" : Real AT %DB4300.DBD10, 500 ms
   "2080AG508M01.AI3" : Real AT %DB4300.DBD14, 500 ms
   "2080AG508M01.AO1a" : Real AT %DB4300.DBD34, 500 ms
   "2080AG508M01.AO1b" : Real AT %DB4300.DBD38, 500 ms
   "2080AG508M01.AO2a" : Real AT %DB4300.DBD42, 500 ms
   "2080AG508M01.AO2b" : Real AT %DB4300.DBD42, 500 ms
   "2080AG508M01.AO3a" : Real AT %DB4300.DBD50, 500 ms
   "2080AG508M01.AO3b" : Real AT %DB4300.DBD46, 500 ms
   "2080AG508M01.BlockInfo" : Array [0..4] of Int AT %DB4300.DBX74.0, 500 ms
   "2080AG508M01.DefaultText" : TextRef, internal   // Заголовок POPUP окна. При експорте из ECS через скрипт заполняется автоматически, если теги копируются в ручную то требуется в ручную задатать свойство Start Value
   "2080AG508M01.DI.ACK" : Bool AT %DB4300.DBX5.3, 500 ms
   "2080AG508M01.DI.ASTR" : Bool AT %DB4300.DBX2.1, 500 ms
   "2080AG508M01.DI.BUSF" : Bool AT %DB4300.DBX4.5, 500 ms
   "2080AG508M01.DI.DIR" : Bool AT %DB4300.DBX2.2, 500 ms
   "2080AG508M01.DI.DOPR" : Bool AT %DB4300.DBX4.6, 500 ms
   "2080AG508M01.DI.DRDY" : Bool AT %DB4300.DBX3.6, 500 ms
   "2080AG508M01.DI.DTEST" : Bool AT %DB4300.DBX4.7, 500 ms
   "2080AG508M01.DI.EARTH" : Bool AT %DB4300.DBX4.1, 500 ms
   "2080AG508M01.DI.ES" : Bool AT %DB4300.DBX5.2, 500 ms
   "2080AG508M01.DI.GFA" : Bool AT %DB4300.DBX4.3, 500 ms
   "2080AG508M01.DI.GWA" : Bool AT %DB4300.DBX4.4, 500 ms
   "2080AG508M01.DI.LSTP" : Bool AT %DB4300.DBX3.2, 500 ms
   "2080AG508M01.DI.LSTR1" : Bool AT %DB4300.DBX3.0, 500 ms
   "2080AG508M01.DI.LSTR2" : Bool AT %DB4300.DBX3.1, 500 ms
   "2080AG508M01.DI.MCC" : Bool AT %DB4300.DBX2.3, 500 ms
   "2080AG508M01.DI.MD" : Bool AT %DB4300.DBX3.7, 500 ms
   "2080AG508M01.DI.OVL" : Bool AT %DB4300.DBX2.5, 500 ms
   "2080AG508M01.DI.RDY" : Bool AT %DB4300.DBX2.4, 500 ms
   "2080AG508M01.DI.REM" : Bool AT %DB4300.DBX3.3, 500 ms
   "2080AG508M01.DI.RET1" : Bool AT %DB4300.DBX2.6, 500 ms
   "2080AG508M01.DI.RET2" : Bool AT %DB4300.DBX2.7, 500 ms
   "2080AG508M01.DI.SEL" : Bool AT %DB4300.DBX2.0, 500 ms
   "2080AG508M01.DI.SFS" : Bool AT %DB4300.DBX5.0, 500 ms
   "2080AG508M01.DI.SLS" : Bool AT %DB4300.DBX5.1, 500 ms
   "2080AG508M01.DI.SSW" : Bool AT %DB4300.DBX3.4, 500 ms
   "2080AG508M01.DI.STALL" : Bool AT %DB4300.DBX4.0, 500 ms
   "2080AG508M01.DI.TFA" : Bool AT %DB4300.DBX3.5, 500 ms
   "2080AG508M01.DI.UBAL" : Bool AT %DB4300.DBX4.2, 500 ms
   "2080AG508M01.DQ.ASTW" : Bool AT %DB4300.DBX32.0, 500 ms
   "2080AG508M01.DQ.AUT" : Bool AT %DB4300.DBX31.4, 500 ms
   "2080AG508M01.DQ.CON1" : Bool AT %DB4300.DBX30.0, 500 ms
   "2080AG508M01.DQ.CON2" : Bool AT %DB4300.DBX30.1, 500 ms
   "2080AG508M01.DQ.LAMP1" : Bool AT %DB4300.DBX30.2, 500 ms
   "2080AG508M01.DQ.LAMP2" : Bool AT %DB4300.DBX30.3, 500 ms
   "2080AG508M01.DQ.LOC" : Bool AT %DB4300.DBX31.2, 500 ms
   "2080AG508M01.DQ.MAN" : Bool AT %DB4300.DBX31.3, 500 ms
   "2080AG508M01.DQ.OK" : Bool AT %DB4300.DBX31.1, 500 ms
   "2080AG508M01.DQ.RD1" : Bool AT %DB4300.DBX30.5, 500 ms
   "2080AG508M01.DQ.RD2" : Bool AT %DB4300.DBX30.6, 500 ms
   "2080AG508M01.DQ.RES" : Bool AT %DB4300.DBX31.6, 500 ms
   "2080AG508M01.DQ.RUN1" : Bool AT %DB4300.DBX30.7, 500 ms
   "2080AG508M01.DQ.RUN2" : Bool AT %DB4300.DBX31.0, 500 ms
   "2080AG508M01.DQ.SACK" : Bool AT %DB4300.DBX30.4, 500 ms
   "2080AG508M01.DQ.SS" : Bool AT %DB4300.DBX31.5, 500 ms
   "2080AG508M01.DQ.TESTP" : Bool AT %DB4300.DBX31.7, 500 ms
   "2080AG508M01.FP_CMD" : Int AT %DB4300.DBW84, 500 ms
   "2080AG508M01.FP_CMD.AckAlarm" : Bool AT %DB4300.DBX84.7, 500 ms
   "2080AG508M01.FP_CMD.Auto" : Bool AT %DB4300.DBX85.0, 500 ms
   "2080AG508M01.FP_CMD.Local" : Bool AT %DB4300.DBX85.2, 500 ms
   "2080AG508M01.FP_CMD.Manual" : Bool AT %DB4300.DBX85.1, 500 ms
   "2080AG508M01.FP_CMD.QuickStop" : Bool AT %DB4300.DBX84.0, 500 ms
   "2080AG508M01.FP_CMD.Reset" : Bool AT %DB4300.DBX85.6, 500 ms
   "2080AG508M01.FP_CMD.Start1" : Bool AT %DB4300.DBX85.3, 500 ms
   "2080AG508M01.FP_CMD.Start2" : Bool AT %DB4300.DBX85.4, 500 ms
   "2080AG508M01.FP_CMD.Stop" : Bool AT %DB4300.DBX85.5, 500 ms
   "2080AG508M01.FP_CMD.Test" : Bool AT %DB4300.DBX85.7, 500 ms
   "2080AG508M01.FP_DIM.Auto" : Bool AT %DB4300.DBX92.0, 500 ms
   "2080AG508M01.FP_DIM.FP_DIM" : Bool AT %DB4300.DBX92.0, 500 ms
   "2080AG508M01.FP_DIM.Local" : Bool AT %DB4300.DBX92.1, 500 ms
   "2080AG508M01.FP_DIM.Manual" : Bool AT %DB4300.DBX92.2, 500 ms
   "2080AG508M01.FP_DIM.QStop" : Bool AT %DB4300.DBX92.7, 500 ms
   "2080AG508M01.FP_DIM.Reset" : Bool AT %DB4300.DBX93.0, 500 ms
   "2080AG508M01.FP_DIM.Start1" : Bool AT %DB4300.DBX92.3, 500 ms
   "2080AG508M01.FP_DIM.Start2" : Bool AT %DB4300.DBX92.4, 500 ms
   "2080AG508M01.FP_DIM.Stop" : Bool AT %DB4300.DBX92.5, 500 ms
   "2080AG508M01.FP_DIM.TEst" : Bool AT %DB4300.DBX92.6, 500 ms
   "2080AG508M01.FP_DIM1" : Array [0..15] of Bool AT %DB4300.DBX92.0, 500 ms
   "2080AG508M01.FP_EN.Mode_Auto" : Bool AT %DB4300.DBX90.0, 500 ms
   "2080AG508M01.FP_EN.Mode_Loc" : Bool AT %DB4300.DBX90.2, 500 ms
   "2080AG508M01.FP_EN.Mode_Loc_1" : Bool AT %DB4300.DBX90.3, 500 ms
   "2080AG508M01.FP_EN.Mode_Man" : Bool AT %DB4300.DBX90.1, 500 ms
   "2080AG508M01.FP_EN.Mode_SS_Field" : Bool AT %DB4300.DBX90.4, 500 ms
   "2080AG508M01.FP_EN.Mode_SS_FP" : Bool AT %DB4300.DBX90.5, 500 ms
   "2080AG508M01.FP_EN.Mode_Test" : Bool AT %DB4300.DBX90.3, 500 ms
   "2080AG508M01.FP_EN.PB_QStop" : Bool AT %DB4300.DBX90.6, 500 ms
   "2080AG508M01.FP_PARM.AI1_Max" : Real AT %DB4300.DBD158, 500 ms
   "2080AG508M01.FP_PARM.AI1_Min" : Real AT %DB4300.DBD162, 500 ms
   "2080AG508M01.FP_PARM.AI2_Max" : Real AT %DB4300.DBD166, 500 ms
   "2080AG508M01.FP_PARM.AI2_Min" : Real AT %DB4300.DBD170, 500 ms
   "2080AG508M01.FP_PARM.AI3_Max" : Real AT %DB4300.DBD174, 500 ms
   "2080AG508M01.FP_PARM.AI3_Min" : Real AT %DB4300.DBD178, 500 ms
   "2080AG508M01.FP_PARM.AO1a_Max" : Real AT %DB4300.DBD182, 500 ms
   "2080AG508M01.FP_PARM.AO1a_Min" : Real AT %DB4300.DBD186, 500 ms
   "2080AG508M01.FP_PARM.AO1b_Max" : Real AT %DB4300.DBD206, 500 ms
   "2080AG508M01.FP_PARM.AO1b_Min" : Real AT %DB4300.DBD210, 500 ms
   "2080AG508M01.FP_PARM.AO2a_Max" : Real AT %DB4300.DBD190, 500 ms
   "2080AG508M01.FP_PARM.AO2a_Min" : Real AT %DB4300.DBD194, 500 ms
   "2080AG508M01.FP_PARM.AO2b_Max" : Real AT %DB4300.DBD214, 500 ms
   "2080AG508M01.FP_PARM.AO2b_Min" : Real AT %DB4300.DBD218, 500 ms
   "2080AG508M01.FP_PARM.AO3a_Max" : Real AT %DB4300.DBD198, 500 ms
   "2080AG508M01.FP_PARM.AO3a_Min" : Real AT %DB4300.DBD202, 500 ms
   "2080AG508M01.FP_PARM.AO3b_Max" : Real AT %DB4300.DBD222, 500 ms
   "2080AG508M01.FP_PARM.AO3b_Min" : Real AT %DB4300.DBD226, 500 ms
   "2080AG508M01.FP_PARM.ChangeDir_Acc" : Int AT %DB4300.DBW138, 500 ms
   "2080AG508M01.FP_PARM.ChangeDir_Pre" : Int AT %DB4300.DBW136, 500 ms
   "2080AG508M01.FP_PARM.DelayStart_Acc" : Int AT %DB4300.DBW114, 500 ms
   "2080AG508M01.FP_PARM.DelayStart_Pre" : Int AT %DB4300.DBW112, 500 ms
   "2080AG508M01.FP_PARM.DelayStop_Acc" : Int AT %DB4300.DBW118, 500 ms
   "2080AG508M01.FP_PARM.DelayStop_Pre" : Int AT %DB4300.DBW116, 500 ms
   "2080AG508M01.FP_PARM.INTL" : Bool AT %DB4300.DBX230.0, 500 ms
   "2080AG508M01.FP_PARM.INTL_SEQ_STP" : Bool AT %DB4300.DBX230.3, 500 ms
   "2080AG508M01.FP_PARM.INTL_SEQ_STR1" : Bool AT %DB4300.DBX230.1, 500 ms
   "2080AG508M01.FP_PARM.INTL_SEQ_STR2" : Bool AT %DB4300.DBX230.2, 500 ms
   "2080AG508M01.FP_PARM.LeaveFS_Acc" : Int AT %DB4300.DBW142, 500 ms
   "2080AG508M01.FP_PARM.LeaveFS_Pre" : Int AT %DB4300.DBW140, 500 ms
   "2080AG508M01.FP_PARM.MD_Freq_PV" : Int AT %DB4300.DBW154, 500 ms
   "2080AG508M01.FP_PARM.MD_Freq_SP" : Int AT %DB4300.DBW152, 500 ms
   "2080AG508M01.FP_PARM.ReachFS_Acc" : Int AT %DB4300.DBW150, 500 ms
   "2080AG508M01.FP_PARM.ReachFS_Pre" : Int AT %DB4300.DBW148, 500 ms
   "2080AG508M01.FP_PARM.ReachLS_Acc" : Int AT %DB4300.DBW146, 500 ms
   "2080AG508M01.FP_PARM.ReachLS_Pre" : Int AT %DB4300.DBW144, 500 ms
   "2080AG508M01.FP_PARM.ReturnMon_Acc" : Int AT %DB4300.DBW122, 500 ms
   "2080AG508M01.FP_PARM.ReturnMon_Pre" : Int AT %DB4300.DBW120, 500 ms
   "2080AG508M01.FP_PARM.RunDelay1_Acc" : Int AT %DB4300.DBW106, 500 ms
   "2080AG508M01.FP_PARM.RunDelay1_Pre" : Int AT %DB4300.DBW104, 500 ms
   "2080AG508M01.FP_PARM.RunDelay2_Acc" : Int AT %DB4300.DBW110, 500 ms
   "2080AG508M01.FP_PARM.RunDelay2_Pre" : Int AT %DB4300.DBW108, 500 ms
   "2080AG508M01.FP_PARM.SpeedMonOffDelay_Acc" : Int AT %DB4300.DBW130, 500 ms
   "2080AG508M01.FP_PARM.SpeedMonOffDelay_Pre" : Int AT %DB4300.DBW128, 500 ms
   "2080AG508M01.FP_PARM.SpeedMonOnDelay_Acc" : Int AT %DB4300.DBW126, 500 ms
   "2080AG508M01.FP_PARM.SpeedMonOnDelay_Pre" : Int AT %DB4300.DBW124, 500 ms
   "2080AG508M01.FP_PARM.SpeedMonTrigDelay_Acc" : Int AT %DB4300.DBW134, 500 ms
   "2080AG508M01.FP_PARM.SpeedMonTrigDelay_Pre" : Int AT %DB4300.DBW132, 500 ms
   "2080AG508M01.FP_PARM.StartWarn_Acc" : Int AT %DB4300.DBW102, 500 ms
   "2080AG508M01.FP_PARM.StartWarn_Pre" : Int AT %DB4300.DBW100, 500 ms
   "2080AG508M01.FP_PARM.StopReason" : Int AT %DB4300.DBW156, 500 ms
   "2080AG508M01.FP_SEL.INCH_Loc" : Bool AT %DB4300.DBX87.7, 500 ms
   "2080AG508M01.FP_SEL.INCH_Man" : Bool AT %DB4300.DBX87.6, 500 ms
   "2080AG508M01.FP_SEL.MD" : Bool AT %DB4300.DBX86.0, 500 ms
   "2080AG508M01.FP_SEL.MD_Maintain" : Bool AT %DB4300.DBX86.3, 500 ms
   "2080AG508M01.FP_SEL.MD_OnOff" : Bool AT %DB4300.DBX86.2, 500 ms
   "2080AG508M01.FP_SEL.MD_Puls" : Bool AT %DB4300.DBX86.1, 500 ms
   "2080AG508M01.FP_SEL.MotorStarter" : Bool AT %DB4300.DBX87.3, 500 ms
   "2080AG508M01.FP_SEL.OutOfSevice" : Bool AT %DB4300.DBX88.0, 500 ms
   "2080AG508M01.FP_SEL.ParentCollection" : Bool AT %DB4300.DBX87.5, 500 ms
   "2080AG508M01.FP_SEL.ParentSupress" : Bool AT %DB4300.DBX87.4, 500 ms
   "2080AG508M01.FP_SEL.STW_AutoStart" : Bool AT %DB4300.DBX86.4, 500 ms
   "2080AG508M01.FP_SEL.STW_Local" : Bool AT %DB4300.DBX86.5, 500 ms
   "2080AG508M01.FP_SEL.STW_Manual" : Bool AT %DB4300.DBX86.6, 500 ms
   "2080AG508M01.FP_SEL.STW_Single" : Bool AT %DB4300.DBX86.7, 500 ms
   "2080AG508M01.FP_SEL.Type_Bimotor" : Bool AT %DB4300.DBX87.1, 500 ms
   "2080AG508M01.FP_SEL.Type_Indication" : Bool AT %DB4300.DBX87.2, 500 ms
   "2080AG508M01.FP_SEL.Type_Unimotor" : Bool AT %DB4300.DBX87.0, 500 ms
   "2080AG508M01.FP_SEL.WarningDrive" : Bool AT %DB4300.DBX88.1, 500 ms
   "2080AG508M01.FP_SHOW.ACK" : Bool AT %DB4300.DBX97.5, 500 ms
   "2080AG508M01.FP_SHOW.AI1" : Bool AT %DB4300.DBX95.0, 500 ms
   "2080AG508M01.FP_SHOW.AI2" : Bool AT %DB4300.DBX95.1, 500 ms
   "2080AG508M01.FP_SHOW.AI3" : Bool AT %DB4300.DBX95.2, 500 ms
   "2080AG508M01.FP_SHOW.ASTR" : Bool AT %DB4300.DBX99.2, 500 ms
   "2080AG508M01.FP_SHOW.B1" : Byte AT %DB4300.DBB95, 500 ms
   "2080AG508M01.FP_SHOW.B2" : Byte AT %DB4300.DBB96, 500 ms
   "2080AG508M01.FP_SHOW.B3" : Byte AT %DB4300.DBB97, 500 ms
   "2080AG508M01.FP_SHOW.B4" : Byte AT %DB4300.DBB98, 500 ms
   "2080AG508M01.FP_SHOW.BUSF" : Bool AT %DB4300.DBX97.2, 500 ms
   "2080AG508M01.FP_SHOW.ChangeDir" : Bool AT %DB4300.DBX99.0, 500 ms
   "2080AG508M01.FP_SHOW.CON2" : Bool AT %DB4300.DBX98.2, 500 ms
   "2080AG508M01.FP_SHOW.DelayRun2" : Bool AT %DB4300.DBX98.7, 500 ms
   "2080AG508M01.FP_SHOW.DOPR" : Bool AT %DB4300.DBX97.3, 500 ms
   "2080AG508M01.FP_SHOW.DRDY" : Bool AT %DB4300.DBX96.4, 500 ms
   "2080AG508M01.FP_SHOW.DTEST" : Bool AT %DB4300.DBX97.4, 500 ms
   "2080AG508M01.FP_SHOW.EARTH" : Bool AT %DB4300.DBX96.6, 500 ms
   "2080AG508M01.FP_SHOW.ES" : Bool AT %DB4300.DBX96.2, 500 ms
   "2080AG508M01.FP_SHOW.GFA" : Bool AT %DB4300.DBX97.0, 500 ms
   "2080AG508M01.FP_SHOW.GWA" : Bool AT %DB4300.DBX97.1, 500 ms
   "2080AG508M01.FP_SHOW.LSTP" : Bool AT %DB4300.DBX95.7, 500 ms
   "2080AG508M01.FP_SHOW.LSTR1" : Bool AT %DB4300.DBX97.6, 500 ms
   "2080AG508M01.FP_SHOW.LSTR2" : Bool AT %DB4300.DBX97.7, 500 ms
   "2080AG508M01.FP_SHOW.MCC" : Bool AT %DB4300.DBX95.4, 500 ms
   "2080AG508M01.FP_SHOW.MD" : Bool AT %DB4300.DBX98.6, 500 ms
   "2080AG508M01.FP_SHOW.OVL" : Bool AT %DB4300.DBX95.6, 500 ms
   "2080AG508M01.FP_SHOW.PB_Auto" : Bool AT %DB4300.DBX94.0, 500 ms
   "2080AG508M01.FP_SHOW.PB_Local" : Bool AT %DB4300.DBX94.1, 500 ms
   "2080AG508M01.FP_SHOW.PB_Manual" : Bool AT %DB4300.DBX94.2, 500 ms
   "2080AG508M01.FP_SHOW.PB_QStop" : Bool AT %DB4300.DBX94.7, 500 ms
   "2080AG508M01.FP_SHOW.PB_Reset" : Bool AT %DB4300.DBX99.1, 500 ms
   "2080AG508M01.FP_SHOW.PB_Start1" : Bool AT %DB4300.DBX94.3, 500 ms
   "2080AG508M01.FP_SHOW.PB_Start2" : Bool AT %DB4300.DBX94.4, 500 ms
   "2080AG508M01.FP_SHOW.PB_Stop" : Bool AT %DB4300.DBX94.5, 500 ms
   "2080AG508M01.FP_SHOW.PB_Test" : Bool AT %DB4300.DBX94.6, 500 ms
   "2080AG508M01.FP_SHOW.RD2" : Bool AT %DB4300.DBX98.3, 500 ms
   "2080AG508M01.FP_SHOW.RDY" : Bool AT %DB4300.DBX95.5, 500 ms
   "2080AG508M01.FP_SHOW.REM" : Bool AT %DB4300.DBX96.0, 500 ms
   "2080AG508M01.FP_SHOW.RET2" : Bool AT %DB4300.DBX98.0, 500 ms
   "2080AG508M01.FP_SHOW.RUN2" : Bool AT %DB4300.DBX98.1, 500 ms
   "2080AG508M01.FP_SHOW.SFS" : Bool AT %DB4300.DBX98.4, 500 ms
   "2080AG508M01.FP_SHOW.SLS" : Bool AT %DB4300.DBX98.5, 500 ms
   "2080AG508M01.FP_SHOW.SP" : Bool AT %DB4300.DBX95.3, 500 ms
   "2080AG508M01.FP_SHOW.SSW" : Bool AT %DB4300.DBX96.1, 500 ms
   "2080AG508M01.FP_SHOW.STALL" : Bool AT %DB4300.DBX96.5, 500 ms
   "2080AG508M01.FP_SHOW.TFA" : Bool AT %DB4300.DBX96.3, 500 ms
   "2080AG508M01.FP_SHOW.UBAL" : Bool AT %DB4300.DBX96.7, 500 ms
   "2080AG508M01.ModePointer" : Int AT %DB4300.DBW496, 500 ms
   "2080AG508M01.MSW" : DWord AT %DB4300.DBD62, 500 ms
   "2080AG508M01.ParentInfo" : TextRef, internal   // Имя родителя для попап окна, вкладка инфо. При експорте из ECS через скрипт заполняется автоматически, если теги копируются в ручную то требуется в ручную задатать свойство Start Value
   "2080AG508M01.SPSET" : Real AT %DB4300.DBD18, 500 ms
   "2080AG508M01.StatusWork" : Int AT %DB4300.DBW494, 500 ms
   "2080AG508M01.STR01" : Byte AT %DB10.DBB389, 500 ms   // Interlock
   "2080AG508M01.STR01.DefaultText" : TextRef, internal

discrete alarms
   1: '', class Errors, trigger "tmp_bool" bit 0

text list "motor_status": 1 'Stopped'; 11..12 'Start Selected'; 21..22 'Start Warn'; 31..32 'Stop Selected'; 41..42 'Stopping'; 45..46 'Wait Start'; 51..52 'Delayed Start'; 61..63 'Interval Start'; 66..67 'Wait Stop'; 71..72 'Delayed Stop'; 81..82 'Running'; 91..92 'Starting'; 99 'Interlocked'; 180 'Test Permission'; 181 'Test Selected'; 190 'Out Of Service'; 200 'Emergency Stop'; 201 'Bus Fault'; 202 'Drawer Pos Fault'; 204 'Drawer Not in Oper.'; 205 'Overload'; 206 'Thermistor Fault'; 207 'Drive Not Ready'; 209 'Not Ready'; 210 'Safety Switch'; 211 'Local Stop Activated'; 212 'Switch Not Remote'; 213 'Motor Stalled'; 214 'Earth Fault'; 215 'Current Unbalance'; 216 'Return Fault'; 217 'Motion Detector Fault'; 218 'Not Leaving 1. Step'; 219 'Not Reach. Last Step'; 220 'Not Back in 1. Step'; 221 'Both 1. and last step'; 222 'Excessive Starts'; 223 'General Fault'; 224 'General Warning'; 225 'MCC Fault'; 300 'No Type Selected'; 301 'Fault State'; 302 'Unknown State'

text list "mode_l": 51 'A'; 52 'M'; 54 'L'; 55 'T'

text list "interlock_status_byte": 0..1 'FLT'; 1 'OK'; 2 'OK Dis'; 3 'OK NA'; 4 'FLT'; 5 'Flt Dis'; 6 'Flt NA'; 7 'OK Invis'; 8 'Flt Invis'

text list "valve_status": 1 'Not Active Midle'; 10..13 'Start Selected'; 14..16 'Wait Start'; 20..23 'Start Warning'; 28 'Start Warn. Park'; 30..33 'Stop Selected'; 40 'Stopping'; 51 'Moving To Open'; 54 'Limit Drifting'; 60 'Interval Start'; 61 'Pos. Open'; 64 'No Position'; 65..67 'Wait Stop'; 70..76 'Delayed Start'; 99 'Interlocked'; 131..133 'Parking'; 180 'Test Permission'; 181 'Test Selected'; 190 'Out Of Service'; 200 'Emergency Stop'; 201 'Bus Fault'; 203 'Test Position'; 205 'Overload'; 207 'Drive Not Ready'; 208 'Not Ready'; 210 'Safety Switch'; 212 'Switch Not Remote'; 223 'General Fault'; 224 'General Warning'; 230 'More Limit On'; 232 'Runtime Fault'; 244 'Limit Drift Alarm'; 302 'No Type Selected'; 303 'Fault State'; 304 'Unknown State'; 63 'Pos. Midle'; 62 'Pos. Close'; 53 'Moving To Midle'; 52 'Moving To Close'; 3 'Not Active Close'; 2 'Not Active Open'; 4 'Not Active'

text list "analog_status": 1 'Normal'; 50 'Activate Block Alarm'; 51 'Activate Advisory Alarm'; 52 'Activate Critical Alarm'; 53 'Unacknowledged Block Alarm'; 54 'Unacknowledged Advisory Alarm'; 55 'Unacknowledged Critical Alarm'; 56 'Init Fail Safe'; 57 'Maintenance Required'; 150 'Open Loop'; 151 'Short Circuit'; 152 'Signal Fault'; 153 'Bad'; 154 'Bad - Configuration Error'; 155 'Bad - Not Connected'; 156 'Bad - Device Failure'; 157 'Bad - No Communication'; 158 'Bad - No Communication'; 159 'Bad - Out of service'; 160 'Bad - Non Measured'; 161 'Bad - Maintenance Alarm'; 162 'Bad - Maintenance Demand'; 163 'Uncertain'; 164 'Uncertain - Last Usable'; 165 'Uncertain - Substiture Set'; 166 'Uncertain - Initial Value'; 167 'Uncertain - Sensor Not Accurate'; 168 'Uncertain - EU range exceeded'; 169 'Uncertain - Sub Normal'; 170 'Uncertain - Configuration Error'; 171 'Simulated Value'; 172 'Calibrating'; 173 'H3 Fatal Alarm'; 174 'L3 Fatal Alarm'; 175 'H2 Alarm'; 176 'L2 Alarm'; 177 'H1 Warning'; 178 'L1 Warning'; 179 'Rate of Change'; 180 'Open Loop'; 181 'Short Circuit'

